Staubli VAL3: RobotMotion3.dtx

bool bSignal
bool bTxt1
bool bTxt2
bool bTxt3
bool btrig
public dio fout = {link=fOut0}
public frame FrmDraw = {x=1000, y=-100, fatherId=world[0]}
mdesc mNomSpeed
num l_nInit = 1500
num nNumTotal = 799
num nNumrecord
num nTxtTotal = 2
num n_sTxt
num ndelay = 258.323
public num nnnn
num ntime = 459.89
pointRx pfrmCad[1500]
  [0] = {x=16.915, y=-25.265, z=273.2, rx=-177, ry=0.5, rz=-161.069, fatherId=FrmDraw[0]}
  [1] = {x=15.593, y=-24.767, z=273.202, rx=-177, ry=0.459, rz=-162.61, fatherId=FrmDraw[0]}
  [2] = {x=14.003, y=-24.227, z=273.204, rx=-177, ry=0.41, rz=-164.442, fatherId=FrmDraw[0]}
  [3] = {x=12.409, y=-23.75, z=273.205, rx=-177, ry=0.362, rz=-166.257, fatherId=FrmDraw[0]}
  [4] = {x=10.813, y=-23.335, z=273.207, rx=-177, ry=0.314, rz=-168.059, fatherId=FrmDraw[0]}
  [5] = {x=9.215, y=-22.978, z=273.208, rx=-177, ry=0.267, rz=-169.848, fatherId=FrmDraw[0]}
  [6] = {x=7.615, y=-22.681, z=273.209, rx=-177, ry=0.22, rz=-171.628, fatherId=FrmDraw[0]}
  [7] = {x=6.014, y=-22.441, z=273.209, rx=-177, ry=0.173, rz=-173.399, fatherId=FrmDraw[0]}
  [8] = {x=4.411, y=-22.259, z=273.21, rx=-177, ry=0.127, rz=-175.164, fatherId=FrmDraw[0]}
  [9] = {x=2.807, y=-22.133, z=273.21, rx=-177, ry=0.081, rz=-176.925, fatherId=FrmDraw[0]}
  [10] = {x=1.203, y=-22.063, z=273.211, rx=-177, ry=0.034, rz=-178.683, fatherId=FrmDraw[0]}
  [11] = {x=0.134, y=-22.047, z=273.211, rx=-177, ry=0.004, rz=-179.854, fatherId=FrmDraw[0]}
  [12] = {x=-1.203, y=-22.063, z=273.211, rx=-177, ry=-0.034, rz=178.683, fatherId=FrmDraw[0]}
  [13] = {x=-2.807, y=-22.133, z=273.21, rx=-177, ry=-0.081, rz=176.925, fatherId=FrmDraw[0]}
  [14] = {x=-4.411, y=-22.259, z=273.21, rx=-177, ry=-0.127, rz=175.164, fatherId=FrmDraw[0]}
  [15] = {x=-6.014, y=-22.441, z=273.209, rx=-177, ry=-0.173, rz=173.399, fatherId=FrmDraw[0]}
  [16] = {x=-7.615, y=-22.681, z=273.209, rx=-177, ry=-0.22, rz=171.628, fatherId=FrmDraw[0]}
  [17] = {x=-9.215, y=-22.978, z=273.208, rx=-177, ry=-0.267, rz=169.848, fatherId=FrmDraw[0]}
  [18] = {x=-10.813, y=-23.335, z=273.207, rx=-177, ry=-0.314, rz=168.059, fatherId=FrmDraw[0]}
  [19] = {x=-12.409, y=-23.75, z=273.205, rx=-177, ry=-0.362, rz=166.257, fatherId=FrmDraw[0]}
  [20] = {x=-14.002, y=-24.227, z=273.204, rx=-177, ry=-0.41, rz=164.442, fatherId=FrmDraw[0]}
  [21] = {x=-15.593, y=-24.767, z=273.202, rx=-177, ry=-0.459, rz=162.61, fatherId=FrmDraw[0]}
  [22] = {x=-16.915, y=-25.265, z=273.2, rx=-177, ry=-0.5, rz=161.069, fatherId=FrmDraw[0]}
  [23] = {x=-16.935, y=-25.265, z=270.798, rx=-177, ry=-0.5, rz=161.071, fatherId=FrmDraw[0]}
  [24] = {x=-16.956, y=-25.264, z=268.2, rx=-177, ry=-0.5, rz=161.073, fatherId=FrmDraw[0]}
  [25] = {x=-15.63, y=-24.766, z=268.202, rx=-177, ry=-0.459, rz=162.614, fatherId=FrmDraw[0]}
  [26] = {x=-14.035, y=-24.226, z=268.204, rx=-177, ry=-0.41, rz=164.445, fatherId=FrmDraw[0]}
  [27] = {x=-12.438, y=-23.75, z=268.205, rx=-177, ry=-0.362, rz=166.26, fatherId=FrmDraw[0]}
  [28] = {x=-10.838, y=-23.334, z=268.207, rx=-177, ry=-0.314, rz=168.061, fatherId=FrmDraw[0]}
  [29] = {x=-9.236, y=-22.978, z=268.208, rx=-177, ry=-0.266, rz=169.85, fatherId=FrmDraw[0]}
  [30] = {x=-7.633, y=-22.681, z=268.209, rx=-177, ry=-0.22, rz=171.63, fatherId=FrmDraw[0]}
  [31] = {x=-6.027, y=-22.441, z=268.209, rx=-177, ry=-0.173, rz=173.401, fatherId=FrmDraw[0]}
  [32] = {x=-4.421, y=-22.259, z=268.21, rx=-177, ry=-0.127, rz=175.165, fatherId=FrmDraw[0]}
  [33] = {x=-2.814, y=-22.133, z=268.21, rx=-177, ry=-0.081, rz=176.926, fatherId=FrmDraw[0]}
  [34] = {x=-1.206, y=-22.063, z=268.211, rx=-177, ry=-0.034, rz=178.683, fatherId=FrmDraw[0]}
  [35] = {x=-0.134, y=-22.047, z=268.211, rx=-177, ry=-0.004, rz=179.854, fatherId=FrmDraw[0]}
  [36] = {x=1.206, y=-22.063, z=268.211, rx=-177, ry=0.034, rz=-178.683, fatherId=FrmDraw[0]}
  [37] = {x=2.814, y=-22.133, z=268.21, rx=-177, ry=0.081, rz=-176.926, fatherId=FrmDraw[0]}
  [38] = {x=4.421, y=-22.259, z=268.21, rx=-177, ry=0.127, rz=-175.165, fatherId=FrmDraw[0]}
  [39] = {x=6.027, y=-22.441, z=268.209, rx=-177, ry=0.173, rz=-173.401, fatherId=FrmDraw[0]}
  [40] = {x=7.633, y=-22.681, z=268.209, rx=-177, ry=0.22, rz=-171.63, fatherId=FrmDraw[0]}
  [41] = {x=9.237, y=-22.978, z=268.208, rx=-177, ry=0.266, rz=-169.85, fatherId=FrmDraw[0]}
  [42] = {x=10.838, y=-23.334, z=268.207, rx=-177, ry=0.314, rz=-168.061, fatherId=FrmDraw[0]}
  [43] = {x=12.438, y=-23.75, z=268.205, rx=-177, ry=0.362, rz=-166.26, fatherId=FrmDraw[0]}
  [44] = {x=14.035, y=-24.226, z=268.204, rx=-177, ry=0.41, rz=-164.445, fatherId=FrmDraw[0]}
  [45] = {x=15.63, y=-24.766, z=268.202, rx=-177, ry=0.459, rz=-162.614, fatherId=FrmDraw[0]}
  [46] = {x=16.956, y=-25.264, z=268.2, rx=-177, ry=0.5, rz=-161.073, fatherId=FrmDraw[0]}
  [47] = {x=16.978, y=-25.265, z=265.798, rx=-177, ry=0.5, rz=-161.071, fatherId=FrmDraw[0]}
  [48] = {x=17.003, y=-25.265, z=263.201, rx=-177, ry=0.5, rz=-161.069, fatherId=FrmDraw[0]}
  [49] = {x=15.673, y=-24.767, z=263.202, rx=-177, ry=0.459, rz=-162.61, fatherId=FrmDraw[0]}
  [50] = {x=14.074, y=-24.227, z=263.204, rx=-177, ry=0.41, rz=-164.442, fatherId=FrmDraw[0]}
  [51] = {x=12.472, y=-23.75, z=263.205, rx=-177, ry=0.362, rz=-166.257, fatherId=FrmDraw[0]}
  [52] = {x=10.868, y=-23.335, z=263.207, rx=-177, ry=0.314, rz=-168.059, fatherId=FrmDraw[0]}
  [53] = {x=9.262, y=-22.978, z=263.208, rx=-177, ry=0.267, rz=-169.848, fatherId=FrmDraw[0]}
  [54] = {x=7.653, y=-22.681, z=263.209, rx=-177, ry=0.22, rz=-171.628, fatherId=FrmDraw[0]}
  [55] = {x=6.044, y=-22.441, z=263.209, rx=-177, ry=0.173, rz=-173.399, fatherId=FrmDraw[0]}
  [56] = {x=4.433, y=-22.259, z=263.21, rx=-177, ry=0.127, rz=-175.164, fatherId=FrmDraw[0]}
  [57] = {x=2.821, y=-22.133, z=263.21, rx=-177, ry=0.081, rz=-176.925, fatherId=FrmDraw[0]}
  [58] = {x=1.209, y=-22.063, z=263.211, rx=-177, ry=0.034, rz=-178.683, fatherId=FrmDraw[0]}
  [59] = {x=0.134, y=-22.047, z=263.211, rx=-177, ry=0.004, rz=-179.854, fatherId=FrmDraw[0]}
  [60] = {x=-1.209, y=-22.063, z=263.211, rx=-177, ry=-0.034, rz=178.683, fatherId=FrmDraw[0]}
  [61] = {x=-2.821, y=-22.133, z=263.21, rx=-177, ry=-0.081, rz=176.925, fatherId=FrmDraw[0]}
  [62] = {x=-4.433, y=-22.259, z=263.21, rx=-177, ry=-0.127, rz=175.165, fatherId=FrmDraw[0]}
  [63] = {x=-6.044, y=-22.441, z=263.209, rx=-177, ry=-0.173, rz=173.399, fatherId=FrmDraw[0]}
  [64] = {x=-7.653, y=-22.681, z=263.209, rx=-177, ry=-0.22, rz=171.628, fatherId=FrmDraw[0]}
  [65] = {x=-9.262, y=-22.978, z=263.208, rx=-177, ry=-0.267, rz=169.848, fatherId=FrmDraw[0]}
  [66] = {x=-10.868, y=-23.335, z=263.207, rx=-177, ry=-0.314, rz=168.059, fatherId=FrmDraw[0]}
  [67] = {x=-12.472, y=-23.75, z=263.205, rx=-177, ry=-0.362, rz=166.257, fatherId=FrmDraw[0]}
  [68] = {x=-14.074, y=-24.227, z=263.204, rx=-177, ry=-0.41, rz=164.442, fatherId=FrmDraw[0]}
  [69] = {x=-15.673, y=-24.767, z=263.202, rx=-177, ry=-0.459, rz=162.61, fatherId=FrmDraw[0]}
  [70] = {x=-17.003, y=-25.265, z=263.201, rx=-177, ry=-0.5, rz=161.069, fatherId=FrmDraw[0]}
  [71] = {x=-17.022, y=-25.265, z=260.799, rx=-177, ry=-0.5, rz=161.071, fatherId=FrmDraw[0]}
  [72] = {x=-17.043, y=-25.264, z=258.201, rx=-177, ry=-0.5, rz=161.074, fatherId=FrmDraw[0]}
  [73] = {x=-15.455, y=-24.676, z=258.203, rx=-177, ry=-0.451, rz=162.906, fatherId=FrmDraw[0]}
  [74] = {x=-13.865, y=-24.15, z=258.204, rx=-177, ry=-0.403, rz=164.72, fatherId=FrmDraw[0]}
  [75] = {x=-12.271, y=-23.686, z=258.206, rx=-177, ry=-0.355, rz=166.519, fatherId=FrmDraw[0]}
  [76] = {x=-10.675, y=-23.282, z=258.207, rx=-177, ry=-0.307, rz=168.304, fatherId=FrmDraw[0]}
  [77] = {x=-9.077, y=-22.937, z=258.208, rx=-177, ry=-0.26, rz=170.078, fatherId=FrmDraw[0]}
  [78] = {x=-7.478, y=-22.649, z=258.209, rx=-177, ry=-0.214, rz=171.842, fatherId=FrmDraw[0]}
  [79] = {x=-5.877, y=-22.418, z=258.209, rx=-177, ry=-0.168, rz=173.599, fatherId=FrmDraw[0]}
  [80] = {x=-4.275, y=-22.243, z=258.21, rx=-177, ry=-0.122, rz=175.349, fatherId=FrmDraw[0]}
  [81] = {x=-2.672, y=-22.123, z=258.21, rx=-177, ry=-0.076, rz=177.095, fatherId=FrmDraw[0]}
  [82] = {x=-1.069, y=-22.059, z=258.211, rx=-177, ry=-0.03, rz=178.838, fatherId=FrmDraw[0]}
  [83] = {y=-22.047, z=258.211, rx=-177, rz=180, fatherId=FrmDraw[0]}
  [84] = {x=1.069, y=-22.059, z=258.211, rx=-177, ry=0.03, rz=-178.838, fatherId=FrmDraw[0]}
  [85] = {x=2.672, y=-22.123, z=258.21, rx=-177, ry=0.076, rz=-177.095, fatherId=FrmDraw[0]}
  [86] = {x=4.275, y=-22.243, z=258.21, rx=-177, ry=0.122, rz=-175.349, fatherId=FrmDraw[0]}
  [87] = {x=5.877, y=-22.418, z=258.209, rx=-177, ry=0.168, rz=-173.599, fatherId=FrmDraw[0]}
  [88] = {x=7.478, y=-22.649, z=258.209, rx=-177, ry=0.214, rz=-171.842, fatherId=FrmDraw[0]}
  [89] = {x=9.077, y=-22.937, z=258.208, rx=-177, ry=0.26, rz=-170.078, fatherId=FrmDraw[0]}
  [90] = {x=10.675, y=-23.282, z=258.207, rx=-177, ry=0.307, rz=-168.304, fatherId=FrmDraw[0]}
  [91] = {x=12.271, y=-23.686, z=258.206, rx=-177, ry=0.355, rz=-166.519, fatherId=FrmDraw[0]}
  [92] = {x=13.865, y=-24.15, z=258.204, rx=-177, ry=0.403, rz=-164.72, fatherId=FrmDraw[0]}
  [93] = {x=15.455, y=-24.676, z=258.203, rx=-177, ry=0.451, rz=-162.906, fatherId=FrmDraw[0]}
  [94] = {x=17.043, y=-25.264, z=258.201, rx=-177, ry=0.5, rz=-161.073, fatherId=FrmDraw[0]}
  [95] = {x=17.066, y=-25.265, z=255.799, rx=-177, ry=0.5, rz=-161.072, fatherId=FrmDraw[0]}
  [96] = {x=17.09, y=-25.265, z=253.201, rx=-177, ry=0.5, rz=-161.07, fatherId=FrmDraw[0]}
  [97] = {x=15.763, y=-24.77, z=253.203, rx=-177, ry=0.459, rz=-162.598, fatherId=FrmDraw[0]}
  [98] = {x=14.169, y=-24.234, z=253.204, rx=-177, ry=0.411, rz=-164.416, fatherId=FrmDraw[0]}
  [99] = {x=12.571, y=-23.76, z=253.206, rx=-177, ry=0.363, rz=-166.217, fatherId=FrmDraw[0]}
  [100] = {x=10.971, y=-23.346, z=253.207, rx=-177, ry=0.315, rz=-168.005, fatherId=FrmDraw[0]}
  [101] = {x=9.369, y=-22.991, z=253.208, rx=-177, ry=0.268, rz=-169.781, fatherId=FrmDraw[0]}
  [102] = {x=7.765, y=-22.693, z=253.209, rx=-177, ry=0.222, rz=-171.547, fatherId=FrmDraw[0]}
  [103] = {x=6.16, y=-22.453, z=253.209, rx=-177, ry=0.176, rz=-173.305, fatherId=FrmDraw[0]}
  [104] = {x=4.554, y=-22.268, z=253.21, rx=-177, ry=0.13, rz=-175.057, fatherId=FrmDraw[0]}
  [105] = {x=2.947, y=-22.139, z=253.21, rx=-177, ry=0.084, rz=-176.804, fatherId=FrmDraw[0]}
  [106] = {x=1.34, y=-22.066, z=253.211, rx=-177, ry=0.038, rz=-178.548, fatherId=FrmDraw[0]}
  [107] = {x=0.268, y=-22.048, z=253.211, rx=-177, ry=0.008, rz=-179.71, fatherId=FrmDraw[0]}
  [108] = {x=-1.34, y=-22.066, z=253.211, rx=-177, ry=-0.038, rz=178.548, fatherId=FrmDraw[0]}
  [109] = {x=-2.947, y=-22.139, z=253.21, rx=-177, ry=-0.084, rz=176.804, fatherId=FrmDraw[0]}
  [110] = {x=-4.554, y=-22.268, z=253.21, rx=-177, ry=-0.13, rz=175.057, fatherId=FrmDraw[0]}
  [111] = {x=-6.16, y=-22.453, z=253.209, rx=-177, ry=-0.176, rz=173.305, fatherId=FrmDraw[0]}
  [112] = {x=-7.765, y=-22.693, z=253.209, rx=-177, ry=-0.222, rz=171.547, fatherId=FrmDraw[0]}
  [113] = {x=-9.369, y=-22.991, z=253.208, rx=-177, ry=-0.268, rz=169.781, fatherId=FrmDraw[0]}
  [114] = {x=-10.971, y=-23.346, z=253.207, rx=-177, ry=-0.315, rz=168.005, fatherId=FrmDraw[0]}
  [115] = {x=-12.571, y=-23.76, z=253.206, rx=-177, ry=-0.363, rz=166.217, fatherId=FrmDraw[0]}
  [116] = {x=-14.169, y=-24.234, z=253.204, rx=-177, ry=-0.411, rz=164.416, fatherId=FrmDraw[0]}
  [117] = {x=-15.763, y=-24.77, z=253.203, rx=-177, ry=-0.459, rz=162.598, fatherId=FrmDraw[0]}
  [118] = {x=-17.09, y=-25.265, z=253.201, rx=-177, ry=-0.5, rz=161.07, fatherId=FrmDraw[0]}
  [119] = {x=-17.109, y=-25.265, z=250.799, rx=-177, ry=-0.5, rz=161.071, fatherId=FrmDraw[0]}
  [120] = {x=-17.13, y=-25.264, z=248.201, rx=-177, ry=-0.5, rz=161.074, fatherId=FrmDraw[0]}
  [121] = {x=-15.8, y=-24.769, z=248.203, rx=-177, ry=-0.459, rz=162.602, fatherId=FrmDraw[0]}
  [122] = {x=-14.202, y=-24.234, z=248.204, rx=-177, ry=-0.411, rz=164.419, fatherId=FrmDraw[0]}
  [123] = {x=-12.6, y=-23.76, z=248.206, rx=-177, ry=-0.363, rz=166.22, fatherId=FrmDraw[0]}
  [124] = {x=-10.996, y=-23.346, z=248.207, rx=-177, ry=-0.315, rz=168.007, fatherId=FrmDraw[0]}
  [125] = {x=-9.391, y=-22.99, z=248.208, rx=-177, ry=-0.268, rz=169.783, fatherId=FrmDraw[0]}
  [126] = {x=-7.783, y=-22.693, z=248.209, rx=-177, ry=-0.222, rz=171.549, fatherId=FrmDraw[0]}
  [127] = {x=-6.174, y=-22.453, z=248.209, rx=-177, ry=-0.175, rz=173.306, fatherId=FrmDraw[0]}
  [128] = {x=-4.565, y=-22.268, z=248.21, rx=-177, ry=-0.13, rz=175.058, fatherId=FrmDraw[0]}
  [129] = {x=-2.954, y=-22.139, z=248.21, rx=-177, ry=-0.084, rz=176.804, fatherId=FrmDraw[0]}
  [130] = {x=-1.343, y=-22.066, z=248.211, rx=-177, ry=-0.038, rz=178.548, fatherId=FrmDraw[0]}
  [131] = {y=-22.047, z=248.211, rx=-177, rz=180, fatherId=FrmDraw[0]}
  [132] = {x=1.343, y=-22.066, z=248.211, rx=-177, ry=0.038, rz=-178.548, fatherId=FrmDraw[0]}
  [133] = {x=2.954, y=-22.139, z=248.21, rx=-177, ry=0.084, rz=-176.804, fatherId=FrmDraw[0]}
  [134] = {x=4.565, y=-22.268, z=248.21, rx=-177, ry=0.13, rz=-175.058, fatherId=FrmDraw[0]}
  [135] = {x=6.174, y=-22.453, z=248.209, rx=-177, ry=0.175, rz=-173.306, fatherId=FrmDraw[0]}
  [136] = {x=7.783, y=-22.693, z=248.209, rx=-177, ry=0.222, rz=-171.549, fatherId=FrmDraw[0]}
  [137] = {x=9.391, y=-22.99, z=248.208, rx=-177, ry=0.268, rz=-169.783, fatherId=FrmDraw[0]}
  [138] = {x=10.997, y=-23.346, z=248.207, rx=-177, ry=0.315, rz=-168.007, fatherId=FrmDraw[0]}
  [139] = {x=12.6, y=-23.76, z=248.206, rx=-177, ry=0.363, rz=-166.22, fatherId=FrmDraw[0]}
  [140] = {x=14.202, y=-24.234, z=248.204, rx=-177, ry=0.411, rz=-164.419, fatherId=FrmDraw[0]}
  [141] = {x=15.8, y=-24.769, z=248.203, rx=-177, ry=0.459, rz=-162.602, fatherId=FrmDraw[0]}
  [142] = {x=17.13, y=-25.264, z=248.201, rx=-177, ry=0.5, rz=-161.074, fatherId=FrmDraw[0]}
  [143] = {x=17.153, y=-25.265, z=245.799, rx=-177, ry=0.5, rz=-161.072, fatherId=FrmDraw[0]}
  [144] = {x=17.177, y=-25.265, z=243.201, rx=-177, ry=0.5, rz=-161.07, fatherId=FrmDraw[0]}
  [145] = {x=15.589, y=-24.681, z=243.203, rx=-177, ry=0.451, rz=-162.888, fatherId=FrmDraw[0]}
  [146] = {x=13.998, y=-24.159, z=243.205, rx=-177, ry=0.403, rz=-164.689, fatherId=FrmDraw[0]}
  [147] = {x=12.404, y=-23.697, z=243.206, rx=-177, ry=0.356, rz=-166.474, fatherId=FrmDraw[0]}
  [148] = {x=10.808, y=-23.294, z=243.207, rx=-177, ry=0.309, rz=-168.247, fatherId=FrmDraw[0]}
  [149] = {x=9.21, y=-22.95, z=243.208, rx=-177, ry=0.262, rz=-170.007, fatherId=FrmDraw[0]}
  [150] = {x=7.61, y=-22.661, z=243.209, rx=-177, ry=0.216, rz=-171.759, fatherId=FrmDraw[0]}
  [151] = {x=6.01, y=-22.429, z=243.21, rx=-177, ry=0.17, rz=-173.502, fatherId=FrmDraw[0]}
  [152] = {x=4.408, y=-22.252, z=243.21, rx=-177, ry=0.125, rz=-175.24, fatherId=FrmDraw[0]}
  [153] = {x=2.805, y=-22.13, z=243.21, rx=-177, ry=0.079, rz=-176.973, fatherId=FrmDraw[0]}
  [154] = {x=1.202, y=-22.062, z=243.211, rx=-177, ry=0.034, rz=-178.703, fatherId=FrmDraw[0]}
  [155] = {x=0.134, y=-22.047, z=243.211, rx=-177, ry=0.004, rz=-179.856, fatherId=FrmDraw[0]}
  [156] = {x=-1.202, y=-22.062, z=243.211, rx=-177, ry=-0.034, rz=178.703, fatherId=FrmDraw[0]}
  [157] = {x=-2.805, y=-22.13, z=243.21, rx=-177, ry=-0.079, rz=176.973, fatherId=FrmDraw[0]}
  [158] = {x=-4.408, y=-22.252, z=243.21, rx=-177, ry=-0.125, rz=175.24, fatherId=FrmDraw[0]}
  [159] = {x=-6.01, y=-22.429, z=243.21, rx=-177, ry=-0.17, rz=173.502, fatherId=FrmDraw[0]}
  [160] = {x=-7.61, y=-22.661, z=243.209, rx=-177, ry=-0.216, rz=171.759, fatherId=FrmDraw[0]}
  [161] = {x=-9.21, y=-22.95, z=243.208, rx=-177, ry=-0.262, rz=170.007, fatherId=FrmDraw[0]}
  [162] = {x=-10.808, y=-23.294, z=243.207, rx=-177, ry=-0.309, rz=168.247, fatherId=FrmDraw[0]}
  [163] = {x=-12.404, y=-23.697, z=243.206, rx=-177, ry=-0.356, rz=166.474, fatherId=FrmDraw[0]}
  [164] = {x=-13.998, y=-24.159, z=243.205, rx=-177, ry=-0.403, rz=164.689, fatherId=FrmDraw[0]}
  [165] = {x=-15.589, y=-24.681, z=243.203, rx=-177, ry=-0.451, rz=162.888, fatherId=FrmDraw[0]}
  [166] = {x=-17.177, y=-25.265, z=243.201, rx=-177, ry=-0.5, rz=161.07, fatherId=FrmDraw[0]}
  [167] = {x=-17.197, y=-25.265, z=240.799, rx=-177, ry=-0.5, rz=161.072, fatherId=FrmDraw[0]}
  [168] = {x=-17.218, y=-25.264, z=238.202, rx=-177, ry=-0.5, rz=161.074, fatherId=FrmDraw[0]}
  [169] = {x=-15.625, y=-24.68, z=238.203, rx=-177, ry=-0.451, rz=162.892, fatherId=FrmDraw[0]}
  [170] = {x=-14.03, y=-24.158, z=238.205, rx=-177, ry=-0.403, rz=164.692, fatherId=FrmDraw[0]}
  [171] = {x=-12.433, y=-23.696, z=238.206, rx=-177, ry=-0.356, rz=166.477, fatherId=FrmDraw[0]}
  [172] = {x=-10.833, y=-23.294, z=238.207, rx=-177, ry=-0.309, rz=168.249, fatherId=FrmDraw[0]}
  [173] = {x=-9.231, y=-22.949, z=238.208, rx=-177, ry=-0.262, rz=170.009, fatherId=FrmDraw[0]}
  [174] = {x=-7.628, y=-22.661, z=238.209, rx=-177, ry=-0.216, rz=171.76, fatherId=FrmDraw[0]}
  [175] = {x=-6.023, y=-22.429, z=238.21, rx=-177, ry=-0.17, rz=173.503, fatherId=FrmDraw[0]}
  [176] = {x=-4.418, y=-22.252, z=238.21, rx=-177, ry=-0.125, rz=175.241, fatherId=FrmDraw[0]}
  [177] = {x=-2.812, y=-22.13, z=238.21, rx=-177, ry=-0.079, rz=176.973, fatherId=FrmDraw[0]}
  [178] = {x=-1.205, y=-22.062, z=238.211, rx=-177, ry=-0.034, rz=178.703, fatherId=FrmDraw[0]}
  [179] = {x=-0.134, y=-22.047, z=238.211, rx=-177, ry=-0.004, rz=179.856, fatherId=FrmDraw[0]}
  [180] = {x=1.205, y=-22.062, z=238.211, rx=-177, ry=0.034, rz=-178.703, fatherId=FrmDraw[0]}
  [181] = {x=2.812, y=-22.13, z=238.21, rx=-177, ry=0.079, rz=-176.973, fatherId=FrmDraw[0]}
  [182] = {x=4.418, y=-22.252, z=238.21, rx=-177, ry=0.125, rz=-175.241, fatherId=FrmDraw[0]}
  [183] = {x=6.023, y=-22.429, z=238.21, rx=-177, ry=0.17, rz=-173.503, fatherId=FrmDraw[0]}
  [184] = {x=7.628, y=-22.661, z=238.209, rx=-177, ry=0.216, rz=-171.76, fatherId=FrmDraw[0]}
  [185] = {x=9.231, y=-22.949, z=238.208, rx=-177, ry=0.262, rz=-170.009, fatherId=FrmDraw[0]}
  [186] = {x=10.833, y=-23.294, z=238.207, rx=-177, ry=0.309, rz=-168.249, fatherId=FrmDraw[0]}
  [187] = {x=12.433, y=-23.697, z=238.206, rx=-177, ry=0.356, rz=-166.477, fatherId=FrmDraw[0]}
  [188] = {x=14.03, y=-24.158, z=238.205, rx=-177, ry=0.403, rz=-164.692, fatherId=FrmDraw[0]}
  [189] = {x=15.625, y=-24.68, z=238.203, rx=-177, ry=0.451, rz=-162.892, fatherId=FrmDraw[0]}
  [190] = {x=17.218, y=-25.264, z=238.202, rx=-177, ry=0.5, rz=-161.074, fatherId=FrmDraw[0]}
  [191] = {x=17.24, y=-25.265, z=235.8, rx=-177, ry=0.5, rz=-161.072, fatherId=FrmDraw[0]}
  [192] = {x=17.265, y=-25.265, z=233.202, rx=-177, ry=0.5, rz=-161.07, fatherId=FrmDraw[0]}
  [193] = {x=15.934, y=-24.774, z=233.203, rx=-177, ry=0.46, rz=-162.586, fatherId=FrmDraw[0]}
  [194] = {x=14.335, y=-24.242, z=233.205, rx=-177, ry=0.411, rz=-164.39, fatherId=FrmDraw[0]}
  [195] = {x=12.733, y=-23.77, z=233.206, rx=-177, ry=0.364, rz=-166.178, fatherId=FrmDraw[0]}
  [196] = {x=11.129, y=-23.358, z=233.207, rx=-177, ry=0.317, rz=-167.952, fatherId=FrmDraw[0]}
  [197] = {x=9.524, y=-23.003, z=233.208, rx=-177, ry=0.27, rz=-169.715, fatherId=FrmDraw[0]}
  [198] = {x=7.916, y=-22.706, z=233.209, rx=-177, ry=0.224, rz=-171.467, fatherId=FrmDraw[0]}
  [199] = {x=6.308, y=-22.464, z=233.209, rx=-177, ry=0.178, rz=-173.212, fatherId=FrmDraw[0]}
  [200] = {x=4.698, y=-22.278, z=233.21, rx=-177, ry=0.132, rz=-174.95, fatherId=FrmDraw[0]}
  [201] = {x=3.088, y=-22.147, z=233.21, rx=-177, ry=0.087, rz=-176.684, fatherId=FrmDraw[0]}
  [202] = {x=1.477, y=-22.07, z=233.211, rx=-177, ry=0.042, rz=-178.415, fatherId=FrmDraw[0]}
  [203] = {x=0.134, y=-22.047, z=233.211, rx=-177, ry=0.004, rz=-179.856, fatherId=FrmDraw[0]}
  [204] = {x=-1.477, y=-22.07, z=233.211, rx=-177, ry=-0.042, rz=178.415, fatherId=FrmDraw[0]}
  [205] = {x=-3.088, y=-22.147, z=233.21, rx=-177, ry=-0.087, rz=176.684, fatherId=FrmDraw[0]}
  [206] = {x=-4.698, y=-22.278, z=233.21, rx=-177, ry=-0.132, rz=174.95, fatherId=FrmDraw[0]}
  [207] = {x=-6.308, y=-22.464, z=233.209, rx=-177, ry=-0.178, rz=173.212, fatherId=FrmDraw[0]}
  [208] = {x=-7.916, y=-22.706, z=233.209, rx=-177, ry=-0.224, rz=171.467, fatherId=FrmDraw[0]}
  [209] = {x=-9.524, y=-23.003, z=233.208, rx=-177, ry=-0.27, rz=169.715, fatherId=FrmDraw[0]}
  [210] = {x=-11.129, y=-23.358, z=233.207, rx=-177, ry=-0.317, rz=167.952, fatherId=FrmDraw[0]}
  [211] = {x=-12.733, y=-23.77, z=233.206, rx=-177, ry=-0.364, rz=166.178, fatherId=FrmDraw[0]}
  [212] = {x=-14.335, y=-24.242, z=233.205, rx=-177, ry=-0.411, rz=164.39, fatherId=FrmDraw[0]}
  [213] = {x=-15.934, y=-24.774, z=233.203, rx=-177, ry=-0.46, rz=162.586, fatherId=FrmDraw[0]}
  [214] = {x=-17.265, y=-25.265, z=233.202, rx=-177, ry=-0.5, rz=161.07, fatherId=FrmDraw[0]}
  [215] = {x=-17.284, y=-25.265, z=230.8, rx=-177, ry=-0.5, rz=161.072, fatherId=FrmDraw[0]}
  [216] = {x=-17.305, y=-25.264, z=228.202, rx=-177, ry=-0.5, rz=161.074, fatherId=FrmDraw[0]}
  [217] = {x=-15.971, y=-24.773, z=228.203, rx=-177, ry=-0.459, rz=162.59, fatherId=FrmDraw[0]}
  [218] = {x=-14.368, y=-24.241, z=228.205, rx=-177, ry=-0.411, rz=164.393, fatherId=FrmDraw[0]}
  [219] = {x=-12.762, y=-23.769, z=228.206, rx=-177, ry=-0.364, rz=166.181, fatherId=FrmDraw[0]}
  [220] = {x=-11.155, y=-23.357, z=228.207, rx=-177, ry=-0.317, rz=167.955, fatherId=FrmDraw[0]}
  [221] = {x=-9.545, y=-23.003, z=228.208, rx=-177, ry=-0.27, rz=169.717, fatherId=FrmDraw[0]}
  [222] = {x=-7.934, y=-22.705, z=228.209, rx=-177, ry=-0.224, rz=171.469, fatherId=FrmDraw[0]}
  [223] = {x=-6.322, y=-22.464, z=228.209, rx=-177, ry=-0.178, rz=173.213, fatherId=FrmDraw[0]}
  [224] = {x=-4.709, y=-22.278, z=228.21, rx=-177, ry=-0.132, rz=174.951, fatherId=FrmDraw[0]}
  [225] = {x=-3.095, y=-22.146, z=228.21, rx=-177, ry=-0.087, rz=176.685, fatherId=FrmDraw[0]}
  [226] = {x=-1.48, y=-22.07, z=228.211, rx=-177, ry=-0.042, rz=178.415, fatherId=FrmDraw[0]}
  [227] = {x=-0.135, y=-22.047, z=228.211, rx=-177, ry=-0.004, rz=179.856, fatherId=FrmDraw[0]}
  [228] = {x=1.48, y=-22.07, z=228.211, rx=-177, ry=0.042, rz=-178.415, fatherId=FrmDraw[0]}
  [229] = {x=3.095, y=-22.146, z=228.21, rx=-177, ry=0.087, rz=-176.685, fatherId=FrmDraw[0]}
  [230] = {x=4.709, y=-22.278, z=228.21, rx=-177, ry=0.132, rz=-174.951, fatherId=FrmDraw[0]}
  [231] = {x=6.322, y=-22.464, z=228.209, rx=-177, ry=0.178, rz=-173.213, fatherId=FrmDraw[0]}
  [232] = {x=7.934, y=-22.705, z=228.209, rx=-177, ry=0.224, rz=-171.469, fatherId=FrmDraw[0]}
  [233] = {x=9.545, y=-23.003, z=228.208, rx=-177, ry=0.27, rz=-169.717, fatherId=FrmDraw[0]}
  [234] = {x=11.155, y=-23.357, z=228.207, rx=-177, ry=0.317, rz=-167.955, fatherId=FrmDraw[0]}
  [235] = {x=12.763, y=-23.769, z=228.206, rx=-177, ry=0.364, rz=-166.181, fatherId=FrmDraw[0]}
  [236] = {x=14.368, y=-24.241, z=228.205, rx=-177, ry=0.411, rz=-164.393, fatherId=FrmDraw[0]}
  [237] = {x=15.971, y=-24.773, z=228.203, rx=-177, ry=0.459, rz=-162.59, fatherId=FrmDraw[0]}
  [238] = {x=17.305, y=-25.264, z=228.202, rx=-177, ry=0.5, rz=-161.074, fatherId=FrmDraw[0]}
  [239] = {x=17.328, y=-25.264, z=225.8, rx=-177, ry=0.5, rz=-161.072, fatherId=FrmDraw[0]}
  [240] = {x=17.352, y=-25.265, z=223.202, rx=-177, ry=0.5, rz=-161.07, fatherId=FrmDraw[0]}
  [241] = {x=15.759, y=-24.685, z=223.204, rx=-177, ry=0.452, rz=-162.874, fatherId=FrmDraw[0]}
  [242] = {x=14.163, y=-24.166, z=223.205, rx=-177, ry=0.404, rz=-164.662, fatherId=FrmDraw[0]}
  [243] = {x=12.565, y=-23.707, z=223.206, rx=-177, ry=0.357, rz=-166.434, fatherId=FrmDraw[0]}
  [244] = {x=10.965, y=-23.306, z=223.207, rx=-177, ry=0.31, rz=-168.192, fatherId=FrmDraw[0]}
  [245] = {x=9.364, y=-22.962, z=223.208, rx=-177, ry=0.264, rz=-169.94, fatherId=FrmDraw[0]}
  [246] = {x=7.761, y=-22.673, z=223.209, rx=-177, ry=0.218, rz=-171.678, fatherId=FrmDraw[0]}
  [247] = {x=6.156, y=-22.44, z=223.21, rx=-177, ry=0.173, rz=-173.409, fatherId=FrmDraw[0]}
  [248] = {x=4.551, y=-22.261, z=223.21, rx=-177, ry=0.128, rz=-175.133, fatherId=FrmDraw[0]}
  [249] = {x=2.945, y=-22.137, z=223.21, rx=-177, ry=0.082, rz=-176.853, fatherId=FrmDraw[0]}
  [250] = {x=1.339, y=-22.065, z=223.211, rx=-177, ry=0.037, rz=-178.57, fatherId=FrmDraw[0]}
  [251] = {x=0.268, y=-22.048, z=223.211, rx=-177, ry=0.007, rz=-179.714, fatherId=FrmDraw[0]}
  [252] = {x=-1.339, y=-22.065, z=223.211, rx=-177, ry=-0.037, rz=178.57, fatherId=FrmDraw[0]}
  [253] = {x=-2.945, y=-22.137, z=223.21, rx=-177, ry=-0.082, rz=176.853, fatherId=FrmDraw[0]}
  [254] = {x=-4.551, y=-22.261, z=223.21, rx=-177, ry=-0.128, rz=175.133, fatherId=FrmDraw[0]}
  [255] = {x=-6.156, y=-22.44, z=223.21, rx=-177, ry=-0.173, rz=173.409, fatherId=FrmDraw[0]}
  [256] = {x=-7.761, y=-22.673, z=223.209, rx=-177, ry=-0.218, rz=171.678, fatherId=FrmDraw[0]}
  [257] = {x=-9.364, y=-22.962, z=223.208, rx=-177, ry=-0.264, rz=169.94, fatherId=FrmDraw[0]}
  [258] = {x=-10.965, y=-23.306, z=223.207, rx=-177, ry=-0.31, rz=168.192, fatherId=FrmDraw[0]}
  [259] = {x=-12.565, y=-23.707, z=223.206, rx=-177, ry=-0.357, rz=166.434, fatherId=FrmDraw[0]}
  [260] = {x=-14.163, y=-24.166, z=223.205, rx=-177, ry=-0.404, rz=164.662, fatherId=FrmDraw[0]}
  [261] = {x=-15.759, y=-24.685, z=223.204, rx=-177, ry=-0.452, rz=162.874, fatherId=FrmDraw[0]}
  [262] = {x=-17.352, y=-25.265, z=223.202, rx=-177, ry=-0.5, rz=161.07, fatherId=FrmDraw[0]}
  [263] = {x=-17.371, y=-25.265, z=220.8, rx=-177, ry=-0.5, rz=161.072, fatherId=FrmDraw[0]}
  [264] = {x=-17.392, y=-25.264, z=218.202, rx=-177, ry=-0.5, rz=161.074, fatherId=FrmDraw[0]}
  [265] = {x=-15.795, y=-24.684, z=218.204, rx=-177, ry=-0.452, rz=162.878, fatherId=FrmDraw[0]}
  [266] = {x=-14.196, y=-24.166, z=218.205, rx=-177, ry=-0.404, rz=164.665, fatherId=FrmDraw[0]}
  [267] = {x=-12.594, y=-23.706, z=218.206, rx=-177, ry=-0.357, rz=166.436, fatherId=FrmDraw[0]}
  [268] = {x=-10.99, y=-23.305, z=218.207, rx=-177, ry=-0.31, rz=168.195, fatherId=FrmDraw[0]}
  [269] = {x=-9.385, y=-22.961, z=218.208, rx=-177, ry=-0.264, rz=169.942, fatherId=FrmDraw[0]}
  [270] = {x=-7.778, y=-22.673, z=218.209, rx=-177, ry=-0.218, rz=171.68, fatherId=FrmDraw[0]}
  [271] = {x=-6.17, y=-22.44, z=218.21, rx=-177, ry=-0.173, rz=173.41, fatherId=FrmDraw[0]}
  [272] = {x=-4.561, y=-22.261, z=218.21, rx=-177, ry=-0.128, rz=175.134, fatherId=FrmDraw[0]}
  [273] = {x=-2.952, y=-22.137, z=218.21, rx=-177, ry=-0.082, rz=176.854, fatherId=FrmDraw[0]}
  [274] = {x=-1.342, y=-22.065, z=218.211, rx=-177, ry=-0.037, rz=178.57, fatherId=FrmDraw[0]}
  [275] = {y=-22.047, z=218.211, rx=-177, rz=180, fatherId=FrmDraw[0]}
  [276] = {x=1.342, y=-22.065, z=218.211, rx=-177, ry=0.037, rz=-178.57, fatherId=FrmDraw[0]}
  [277] = {x=2.952, y=-22.137, z=218.21, rx=-177, ry=0.082, rz=-176.854, fatherId=FrmDraw[0]}
  [278] = {x=4.561, y=-22.261, z=218.21, rx=-177, ry=0.128, rz=-175.134, fatherId=FrmDraw[0]}
  [279] = {x=6.17, y=-22.44, z=218.21, rx=-177, ry=0.173, rz=-173.41, fatherId=FrmDraw[0]}
  [280] = {x=7.778, y=-22.673, z=218.209, rx=-177, ry=0.218, rz=-171.68, fatherId=FrmDraw[0]}
  [281] = {x=9.385, y=-22.961, z=218.208, rx=-177, ry=0.264, rz=-169.942, fatherId=FrmDraw[0]}
  [282] = {x=10.99, y=-23.305, z=218.207, rx=-177, ry=0.31, rz=-168.195, fatherId=FrmDraw[0]}
  [283] = {x=12.594, y=-23.706, z=218.206, rx=-177, ry=0.357, rz=-166.436, fatherId=FrmDraw[0]}
  [284] = {x=14.196, y=-24.166, z=218.205, rx=-177, ry=0.404, rz=-164.665, fatherId=FrmDraw[0]}
  [285] = {x=15.795, y=-24.684, z=218.204, rx=-177, ry=0.452, rz=-162.878, fatherId=FrmDraw[0]}
  [286] = {x=17.392, y=-25.264, z=218.202, rx=-177, ry=0.5, rz=-161.074, fatherId=FrmDraw[0]}
  [287] = {x=17.415, y=-25.264, z=215.8, rx=-177, ry=0.5, rz=-161.072, fatherId=FrmDraw[0]}
  [288] = {x=17.439, y=-25.265, z=213.203, rx=-177, ry=0.5, rz=-161.07, fatherId=FrmDraw[0]}
  [289] = {x=15.838, y=-24.685, z=213.204, rx=-177, ry=0.452, rz=-162.874, fatherId=FrmDraw[0]}
  [290] = {x=14.234, y=-24.166, z=213.205, rx=-177, ry=0.404, rz=-164.662, fatherId=FrmDraw[0]}
  [291] = {x=12.628, y=-23.707, z=213.206, rx=-177, ry=0.357, rz=-166.434, fatherId=FrmDraw[0]}
  [292] = {x=11.02, y=-23.306, z=213.207, rx=-177, ry=0.31, rz=-168.192, fatherId=FrmDraw[0]}
  [293] = {x=9.41, y=-22.962, z=213.208, rx=-177, ry=0.264, rz=-169.94, fatherId=FrmDraw[0]}
  [294] = {x=7.799, y=-22.673, z=213.209, rx=-177, ry=0.218, rz=-171.678, fatherId=FrmDraw[0]}
  [295] = {x=6.186, y=-22.44, z=213.21, rx=-177, ry=0.173, rz=-173.409, fatherId=FrmDraw[0]}
  [296] = {x=4.573, y=-22.261, z=213.21, rx=-177, ry=0.128, rz=-175.133, fatherId=FrmDraw[0]}
  [297] = {x=2.959, y=-22.137, z=213.21, rx=-177, ry=0.082, rz=-176.853, fatherId=FrmDraw[0]}
  [298] = {x=1.345, y=-22.065, z=213.211, rx=-177, ry=0.037, rz=-178.57, fatherId=FrmDraw[0]}
  [299] = {x=0.269, y=-22.048, z=213.211, rx=-177, ry=0.007, rz=-179.714, fatherId=FrmDraw[0]}
  [300] = {x=-1.345, y=-22.065, z=213.211, rx=-177, ry=-0.037, rz=178.57, fatherId=FrmDraw[0]}
  [301] = {x=-2.959, y=-22.137, z=213.21, rx=-177, ry=-0.082, rz=176.853, fatherId=FrmDraw[0]}
  [302] = {x=-4.573, y=-22.261, z=213.21, rx=-177, ry=-0.128, rz=175.133, fatherId=FrmDraw[0]}
  [303] = {x=-6.186, y=-22.44, z=213.21, rx=-177, ry=-0.173, rz=173.409, fatherId=FrmDraw[0]}
  [304] = {x=-7.799, y=-22.673, z=213.209, rx=-177, ry=-0.218, rz=171.678, fatherId=FrmDraw[0]}
  [305] = {x=-9.41, y=-22.962, z=213.208, rx=-177, ry=-0.264, rz=169.94, fatherId=FrmDraw[0]}
  [306] = {x=-11.02, y=-23.306, z=213.207, rx=-177, ry=-0.31, rz=168.192, fatherId=FrmDraw[0]}
  [307] = {x=-12.628, y=-23.707, z=213.206, rx=-177, ry=-0.357, rz=166.434, fatherId=FrmDraw[0]}
  [308] = {x=-14.234, y=-24.166, z=213.205, rx=-177, ry=-0.404, rz=164.662, fatherId=FrmDraw[0]}
  [309] = {x=-15.838, y=-24.685, z=213.204, rx=-177, ry=-0.452, rz=162.874, fatherId=FrmDraw[0]}
  [310] = {x=-17.439, y=-25.265, z=213.203, rx=-177, ry=-0.5, rz=161.07, fatherId=FrmDraw[0]}
  [311] = {x=-17.459, y=-25.264, z=210.801, rx=-177, ry=-0.5, rz=161.072, fatherId=FrmDraw[0]}
  [312] = {x=-17.48, y=-25.264, z=208.203, rx=-177, ry=-0.5, rz=161.074, fatherId=FrmDraw[0]}
  [313] = {x=-16.142, y=-24.776, z=208.204, rx=-177, ry=-0.46, rz=162.579, fatherId=FrmDraw[0]}
  [314] = {x=-14.535, y=-24.248, z=208.205, rx=-177, ry=-0.412, rz=164.368, fatherId=FrmDraw[0]}
  [315] = {x=-12.925, y=-23.779, z=208.206, rx=-177, ry=-0.365, rz=166.142, fatherId=FrmDraw[0]}
  [316] = {x=-11.313, y=-23.368, z=208.207, rx=-177, ry=-0.318, rz=167.903, fatherId=FrmDraw[0]}
  [317] = {x=-9.7, y=-23.015, z=208.208, rx=-177, ry=-0.272, rz=169.652, fatherId=FrmDraw[0]}
  [318] = {x=-8.085, y=-22.717, z=208.209, rx=-177, ry=-0.226, rz=171.391, fatherId=FrmDraw[0]}
  [319] = {x=-6.47, y=-22.475, z=208.21, rx=-177, ry=-0.18, rz=173.122, fatherId=FrmDraw[0]}
  [320] = {x=-4.853, y=-22.287, z=208.21, rx=-177, ry=-0.135, rz=174.847, fatherId=FrmDraw[0]}
  [321] = {x=-3.236, y=-22.154, z=208.21, rx=-177, ry=-0.09, rz=176.567, fatherId=FrmDraw[0]}
  [322] = {x=-1.618, y=-22.074, z=208.211, rx=-177, ry=-0.045, rz=178.284, fatherId=FrmDraw[0]}
  [323] = {y=-22.047, z=208.211, rx=-177, rz=180, fatherId=FrmDraw[0]}
  [324] = {x=1.618, y=-22.074, z=208.211, rx=-177, ry=0.045, rz=-178.284, fatherId=FrmDraw[0]}
  [325] = {x=3.236, y=-22.154, z=208.21, rx=-177, ry=0.09, rz=-176.567, fatherId=FrmDraw[0]}
  [326] = {x=4.853, y=-22.287, z=208.21, rx=-177, ry=0.135, rz=-174.847, fatherId=FrmDraw[0]}
  [327] = {x=6.47, y=-22.475, z=208.21, rx=-177, ry=0.18, rz=-173.122, fatherId=FrmDraw[0]}
  [328] = {x=8.085, y=-22.717, z=208.209, rx=-177, ry=0.226, rz=-171.391, fatherId=FrmDraw[0]}
  [329] = {x=9.7, y=-23.015, z=208.208, rx=-177, ry=0.272, rz=-169.651, fatherId=FrmDraw[0]}
  [330] = {x=11.313, y=-23.368, z=208.207, rx=-177, ry=0.318, rz=-167.902, fatherId=FrmDraw[0]}
  [331] = {x=12.925, y=-23.779, z=208.206, rx=-177, ry=0.365, rz=-166.142, fatherId=FrmDraw[0]}
  [332] = {x=14.535, y=-24.248, z=208.205, rx=-177, ry=0.412, rz=-164.368, fatherId=FrmDraw[0]}
  [333] = {x=16.142, y=-24.776, z=208.204, rx=-177, ry=0.46, rz=-162.579, fatherId=FrmDraw[0]}
  [334] = {x=17.48, y=-25.264, z=208.203, rx=-177, ry=0.5, rz=-161.074, fatherId=FrmDraw[0]}
  [335] = {x=17.502, y=-25.264, z=205.801, rx=-177, ry=0.5, rz=-161.072, fatherId=FrmDraw[0]}
  [336] = {x=17.527, y=-25.265, z=203.203, rx=-177, ry=0.5, rz=-161.07, fatherId=FrmDraw[0]}
  [337] = {x=15.929, y=-24.689, z=203.204, rx=-177, ry=0.452, rz=-162.861, fatherId=FrmDraw[0]}
  [338] = {x=14.329, y=-24.174, z=203.206, rx=-177, ry=0.405, rz=-164.635, fatherId=FrmDraw[0]}
  [339] = {x=12.727, y=-23.717, z=203.207, rx=-177, ry=0.358, rz=-166.393, fatherId=FrmDraw[0]}
  [340] = {x=11.123, y=-23.317, z=203.208, rx=-177, ry=0.312, rz=-168.139, fatherId=FrmDraw[0]}
  [341] = {x=9.518, y=-22.974, z=203.208, rx=-177, ry=0.266, rz=-169.874, fatherId=FrmDraw[0]}
  [342] = {x=7.911, y=-22.685, z=203.209, rx=-177, ry=0.22, rz=-171.599, fatherId=FrmDraw[0]}
  [343] = {x=6.303, y=-22.451, z=203.21, rx=-177, ry=0.175, rz=-173.316, fatherId=FrmDraw[0]}
  [344] = {x=4.695, y=-22.271, z=203.21, rx=-177, ry=0.13, rz=-175.028, fatherId=FrmDraw[0]}
  [345] = {x=3.085, y=-22.144, z=203.21, rx=-177, ry=0.086, rz=-176.735, fatherId=FrmDraw[0]}
  [346] = {x=1.476, y=-22.069, z=203.211, rx=-177, ry=0.041, rz=-178.439, fatherId=FrmDraw[0]}
  [347] = {x=0.134, y=-22.047, z=203.211, rx=-177, ry=0.004, rz=-179.858, fatherId=FrmDraw[0]}
  [348] = {x=-1.476, y=-22.069, z=203.211, rx=-177, ry=-0.041, rz=178.439, fatherId=FrmDraw[0]}
  [349] = {x=-3.085, y=-22.144, z=203.21, rx=-177, ry=-0.086, rz=176.735, fatherId=FrmDraw[0]}
  [350] = {x=-4.695, y=-22.271, z=203.21, rx=-177, ry=-0.13, rz=175.028, fatherId=FrmDraw[0]}
  [351] = {x=-6.303, y=-22.451, z=203.21, rx=-177, ry=-0.175, rz=173.316, fatherId=FrmDraw[0]}
  [352] = {x=-7.911, y=-22.685, z=203.209, rx=-177, ry=-0.22, rz=171.599, fatherId=FrmDraw[0]}
  [353] = {x=-9.518, y=-22.974, z=203.208, rx=-177, ry=-0.266, rz=169.874, fatherId=FrmDraw[0]}
  [354] = {x=-11.123, y=-23.317, z=203.208, rx=-177, ry=-0.312, rz=168.139, fatherId=FrmDraw[0]}
  [355] = {x=-12.727, y=-23.717, z=203.207, rx=-177, ry=-0.358, rz=166.393, fatherId=FrmDraw[0]}
  [356] = {x=-14.329, y=-24.174, z=203.206, rx=-177, ry=-0.405, rz=164.635, fatherId=FrmDraw[0]}
  [357] = {x=-15.929, y=-24.689, z=203.204, rx=-177, ry=-0.452, rz=162.861, fatherId=FrmDraw[0]}
  [358] = {x=-17.527, y=-25.265, z=203.203, rx=-177, ry=-0.5, rz=161.07, fatherId=FrmDraw[0]}
  [359] = {x=-17.546, y=-25.264, z=200.801, rx=-177, ry=-0.5, rz=161.072, fatherId=FrmDraw[0]}
  [360] = {x=-17.567, y=-25.264, z=198.203, rx=-177, ry=-0.5, rz=161.074, fatherId=FrmDraw[0]}
  [361] = {x=-15.966, y=-24.688, z=198.204, rx=-177, ry=-0.452, rz=162.864, fatherId=FrmDraw[0]}
  [362] = {x=-14.362, y=-24.173, z=198.206, rx=-177, ry=-0.405, rz=164.638, fatherId=FrmDraw[0]}
  [363] = {x=-12.756, y=-23.716, z=198.207, rx=-177, ry=-0.358, rz=166.396, fatherId=FrmDraw[0]}
  [364] = {x=-11.148, y=-23.317, z=198.208, rx=-177, ry=-0.312, rz=168.141, fatherId=FrmDraw[0]}
  [365] = {x=-9.539, y=-22.973, z=198.208, rx=-177, ry=-0.266, rz=169.876, fatherId=FrmDraw[0]}
  [366] = {x=-7.929, y=-22.685, z=198.209, rx=-177, ry=-0.22, rz=171.6, fatherId=FrmDraw[0]}
  [367] = {x=-6.317, y=-22.451, z=198.21, rx=-177, ry=-0.175, rz=173.318, fatherId=FrmDraw[0]}
  [368] = {x=-4.705, y=-22.271, z=198.21, rx=-177, ry=-0.13, rz=175.029, fatherId=FrmDraw[0]}
  [369] = {x=-3.092, y=-22.143, z=198.21, rx=-177, ry=-0.086, rz=176.736, fatherId=FrmDraw[0]}
  [370] = {x=-1.479, y=-22.069, z=198.211, rx=-177, ry=-0.041, rz=178.439, fatherId=FrmDraw[0]}
  [371] = {x=-0.134, y=-22.047, z=198.211, rx=-177, ry=-0.004, rz=179.858, fatherId=FrmDraw[0]}
  [372] = {x=1.479, y=-22.069, z=198.211, rx=-177, ry=0.041, rz=-178.439, fatherId=FrmDraw[0]}
  [373] = {x=3.092, y=-22.143, z=198.21, rx=-177, ry=0.086, rz=-176.736, fatherId=FrmDraw[0]}
  [374] = {x=4.705, y=-22.271, z=198.21, rx=-177, ry=0.13, rz=-175.029, fatherId=FrmDraw[0]}
  [375] = {x=6.317, y=-22.451, z=198.21, rx=-177, ry=0.175, rz=-173.318, fatherId=FrmDraw[0]}
  [376] = {x=7.929, y=-22.685, z=198.209, rx=-177, ry=0.22, rz=-171.6, fatherId=FrmDraw[0]}
  [377] = {x=9.539, y=-22.973, z=198.208, rx=-177, ry=0.266, rz=-169.875, fatherId=FrmDraw[0]}
  [378] = {x=11.148, y=-23.317, z=198.208, rx=-177, ry=0.312, rz=-168.141, fatherId=FrmDraw[0]}
  [379] = {x=12.756, y=-23.716, z=198.207, rx=-177, ry=0.358, rz=-166.396, fatherId=FrmDraw[0]}
  [380] = {x=14.362, y=-24.173, z=198.206, rx=-177, ry=0.405, rz=-164.638, fatherId=FrmDraw[0]}
  [381] = {x=15.966, y=-24.688, z=198.204, rx=-177, ry=0.452, rz=-162.864, fatherId=FrmDraw[0]}
  [382] = {x=17.567, y=-25.264, z=198.203, rx=-177, ry=0.5, rz=-161.074, fatherId=FrmDraw[0]}
  [383] = {x=17.59, y=-25.264, z=195.801, rx=-177, ry=0.5, rz=-161.072, fatherId=FrmDraw[0]}
  [384] = {x=17.614, y=-25.265, z=193.203, rx=-177, ry=0.5, rz=-161.07, fatherId=FrmDraw[0]}
  [385] = {x=16.008, y=-24.689, z=193.205, rx=-177, ry=0.452, rz=-162.861, fatherId=FrmDraw[0]}
  [386] = {x=14.4, y=-24.174, z=193.206, rx=-177, ry=0.405, rz=-164.635, fatherId=FrmDraw[0]}
  [387] = {x=12.79, y=-23.717, z=193.207, rx=-177, ry=0.358, rz=-166.393, fatherId=FrmDraw[0]}
  [388] = {x=11.178, y=-23.317, z=193.208, rx=-177, ry=0.312, rz=-168.139, fatherId=FrmDraw[0]}
  [389] = {x=9.564, y=-22.974, z=193.209, rx=-177, ry=0.266, rz=-169.874, fatherId=FrmDraw[0]}
  [390] = {x=7.949, y=-22.685, z=193.209, rx=-177, ry=0.22, rz=-171.599, fatherId=FrmDraw[0]}
  [391] = {x=6.334, y=-22.451, z=193.21, rx=-177, ry=0.175, rz=-173.316, fatherId=FrmDraw[0]}
  [392] = {x=4.717, y=-22.271, z=193.21, rx=-177, ry=0.13, rz=-175.028, fatherId=FrmDraw[0]}
  [393] = {x=3.1, y=-22.143, z=193.21, rx=-177, ry=0.086, rz=-176.735, fatherId=FrmDraw[0]}
  [394] = {x=1.483, y=-22.069, z=193.211, rx=-177, ry=0.041, rz=-178.439, fatherId=FrmDraw[0]}
  [395] = {x=0.135, y=-22.047, z=193.211, rx=-177, ry=0.004, rz=-179.858, fatherId=FrmDraw[0]}
  [396] = {x=-1.483, y=-22.069, z=193.211, rx=-177, ry=-0.041, rz=178.439, fatherId=FrmDraw[0]}
  [397] = {x=-3.1, y=-22.144, z=193.21, rx=-177, ry=-0.086, rz=176.735, fatherId=FrmDraw[0]}
  [398] = {x=-4.717, y=-22.271, z=193.21, rx=-177, ry=-0.13, rz=175.028, fatherId=FrmDraw[0]}
  [399] = {x=-6.334, y=-22.451, z=193.21, rx=-177, ry=-0.175, rz=173.316, fatherId=FrmDraw[0]}
  [400] = {x=-7.949, y=-22.685, z=193.209, rx=-177, ry=-0.22, rz=171.599, fatherId=FrmDraw[0]}
  [401] = {x=-9.564, y=-22.974, z=193.209, rx=-177, ry=-0.266, rz=169.874, fatherId=FrmDraw[0]}
  [402] = {x=-11.178, y=-23.317, z=193.208, rx=-177, ry=-0.312, rz=168.139, fatherId=FrmDraw[0]}
  [403] = {x=-12.79, y=-23.717, z=193.207, rx=-177, ry=-0.358, rz=166.393, fatherId=FrmDraw[0]}
  [404] = {x=-14.4, y=-24.174, z=193.206, rx=-177, ry=-0.405, rz=164.635, fatherId=FrmDraw[0]}
  [405] = {x=-16.008, y=-24.689, z=193.205, rx=-177, ry=-0.452, rz=162.861, fatherId=FrmDraw[0]}
  [406] = {x=-17.614, y=-25.265, z=193.203, rx=-177, ry=-0.5, rz=161.07, fatherId=FrmDraw[0]}
  [407] = {x=-17.633, y=-25.264, z=190.801, rx=-177, ry=-0.5, rz=161.072, fatherId=FrmDraw[0]}
  [408] = {x=-17.654, y=-25.264, z=188.204, rx=-177, ry=-0.5, rz=161.074, fatherId=FrmDraw[0]}
  [409] = {x=-16.057, y=-24.692, z=188.205, rx=-177, ry=-0.452, rz=162.851, fatherId=FrmDraw[0]}
  [410] = {x=-14.457, y=-24.18, z=188.206, rx=-177, ry=-0.405, rz=164.611, fatherId=FrmDraw[0]}
  [411] = {x=-12.855, y=-23.726, z=188.207, rx=-177, ry=-0.359, rz=166.356, fatherId=FrmDraw[0]}
  [412] = {x=-11.252, y=-23.328, z=188.208, rx=-177, ry=-0.313, rz=168.089, fatherId=FrmDraw[0]}
  [413] = {x=-9.647, y=-22.985, z=188.209, rx=-177, ry=-0.268, rz=169.81, fatherId=FrmDraw[0]}
  [414] = {x=-8.041, y=-22.697, z=188.209, rx=-177, ry=-0.222, rz=171.522, fatherId=FrmDraw[0]}
  [415] = {x=-6.434, y=-22.462, z=188.21, rx=-177, ry=-0.178, rz=173.227, fatherId=FrmDraw[0]}
  [416] = {x=-4.826, y=-22.28, z=188.21, rx=-177, ry=-0.133, rz=174.925, fatherId=FrmDraw[0]}
  [417] = {x=-3.218, y=-22.15, z=188.21, rx=-177, ry=-0.089, rz=176.619, fatherId=FrmDraw[0]}
  [418] = {x=-1.609, y=-22.073, z=188.211, rx=-177, ry=-0.044, rz=178.31, fatherId=FrmDraw[0]}
  [419] = {y=-22.047, z=188.211, rx=-177, rz=180, fatherId=FrmDraw[0]}
  [420] = {x=1.609, y=-22.073, z=188.211, rx=-177, ry=0.044, rz=-178.31, fatherId=FrmDraw[0]}
  [421] = {x=3.218, y=-22.15, z=188.21, rx=-177, ry=0.089, rz=-176.619, fatherId=FrmDraw[0]}
  [422] = {x=4.826, y=-22.28, z=188.21, rx=-177, ry=0.133, rz=-174.925, fatherId=FrmDraw[0]}
  [423] = {x=6.434, y=-22.462, z=188.21, rx=-177, ry=0.178, rz=-173.227, fatherId=FrmDraw[0]}
  [424] = {x=8.041, y=-22.697, z=188.209, rx=-177, ry=0.222, rz=-171.522, fatherId=FrmDraw[0]}
  [425] = {x=9.647, y=-22.985, z=188.209, rx=-177, ry=0.268, rz=-169.81, fatherId=FrmDraw[0]}
  [426] = {x=11.252, y=-23.328, z=188.208, rx=-177, ry=0.313, rz=-168.089, fatherId=FrmDraw[0]}
  [427] = {x=12.855, y=-23.726, z=188.207, rx=-177, ry=0.359, rz=-166.356, fatherId=FrmDraw[0]}
  [428] = {x=14.457, y=-24.18, z=188.206, rx=-177, ry=0.405, rz=-164.611, fatherId=FrmDraw[0]}
  [429] = {x=16.057, y=-24.692, z=188.205, rx=-177, ry=0.452, rz=-162.851, fatherId=FrmDraw[0]}
  [430] = {x=17.654, y=-25.264, z=188.204, rx=-177, ry=0.5, rz=-161.074, fatherId=FrmDraw[0]}
  [431] = {x=17.677, y=-25.264, z=185.801, rx=-177, ry=0.5, rz=-161.072, fatherId=FrmDraw[0]}
  [432] = {x=17.702, y=-25.265, z=183.204, rx=-177, ry=0.5, rz=-161.07, fatherId=FrmDraw[0]}
  [433] = {x=16.099, y=-24.693, z=183.205, rx=-177, ry=0.453, rz=-162.847, fatherId=FrmDraw[0]}
  [434] = {x=14.495, y=-24.181, z=183.206, rx=-177, ry=0.406, rz=-164.608, fatherId=FrmDraw[0]}
  [435] = {x=12.889, y=-23.727, z=183.207, rx=-177, ry=0.359, rz=-166.354, fatherId=FrmDraw[0]}
  [436] = {x=11.281, y=-23.329, z=183.208, rx=-177, ry=0.313, rz=-168.086, fatherId=FrmDraw[0]}
  [437] = {x=9.672, y=-22.986, z=183.209, rx=-177, ry=0.268, rz=-169.808, fatherId=FrmDraw[0]}
  [438] = {x=8.062, y=-22.697, z=183.209, rx=-177, ry=0.222, rz=-171.521, fatherId=FrmDraw[0]}
  [439] = {x=6.45, y=-22.462, z=183.21, rx=-177, ry=0.178, rz=-173.225, fatherId=FrmDraw[0]}
  [440] = {x=4.839, y=-22.28, z=183.21, rx=-177, ry=0.133, rz=-174.924, fatherId=FrmDraw[0]}
  [441] = {x=3.226, y=-22.151, z=183.21, rx=-177, ry=0.089, rz=-176.619, fatherId=FrmDraw[0]}
  [442] = {x=1.613, y=-22.073, z=183.211, rx=-177, ry=0.044, rz=-178.31, fatherId=FrmDraw[0]}
  [443] = {y=-22.047, z=183.211, rx=-177, rz=180, fatherId=FrmDraw[0]}
  [444] = {x=-1.613, y=-22.073, z=183.211, rx=-177, ry=-0.044, rz=178.31, fatherId=FrmDraw[0]}
  [445] = {x=-3.226, y=-22.151, z=183.21, rx=-177, ry=-0.089, rz=176.619, fatherId=FrmDraw[0]}
  [446] = {x=-4.838, y=-22.28, z=183.21, rx=-177, ry=-0.133, rz=174.924, fatherId=FrmDraw[0]}
  [447] = {x=-6.45, y=-22.462, z=183.21, rx=-177, ry=-0.178, rz=173.225, fatherId=FrmDraw[0]}
  [448] = {x=-8.062, y=-22.697, z=183.209, rx=-177, ry=-0.222, rz=171.521, fatherId=FrmDraw[0]}
  [449] = {x=-9.672, y=-22.986, z=183.209, rx=-177, ry=-0.268, rz=169.808, fatherId=FrmDraw[0]}
  [450] = {x=-11.281, y=-23.329, z=183.208, rx=-177, ry=-0.313, rz=168.086, fatherId=FrmDraw[0]}
  [451] = {x=-12.889, y=-23.727, z=183.207, rx=-177, ry=-0.359, rz=166.354, fatherId=FrmDraw[0]}
  [452] = {x=-14.495, y=-24.181, z=183.206, rx=-177, ry=-0.406, rz=164.608, fatherId=FrmDraw[0]}
  [453] = {x=-16.099, y=-24.693, z=183.205, rx=-177, ry=-0.453, rz=162.847, fatherId=FrmDraw[0]}
  [454] = {x=-17.701, y=-25.265, z=183.204, rx=-177, ry=-0.5, rz=161.07, fatherId=FrmDraw[0]}
  [455] = {x=-17.721, y=-25.264, z=180.802, rx=-177, ry=-0.5, rz=161.072, fatherId=FrmDraw[0]}
  [456] = {x=-17.742, y=-25.264, z=178.204, rx=-177, ry=-0.5, rz=161.074, fatherId=FrmDraw[0]}
  [457] = {x=-16.136, y=-24.692, z=178.205, rx=-177, ry=-0.452, rz=162.851, fatherId=FrmDraw[0]}
  [458] = {x=-14.528, y=-24.18, z=178.206, rx=-177, ry=-0.405, rz=164.611, fatherId=FrmDraw[0]}
  [459] = {x=-12.918, y=-23.726, z=178.207, rx=-177, ry=-0.359, rz=166.356, fatherId=FrmDraw[0]}
  [460] = {x=-11.306, y=-23.328, z=178.208, rx=-177, ry=-0.313, rz=168.089, fatherId=FrmDraw[0]}
  [461] = {x=-9.693, y=-22.985, z=178.209, rx=-177, ry=-0.268, rz=169.81, fatherId=FrmDraw[0]}
  [462] = {x=-8.08, y=-22.697, z=178.209, rx=-177, ry=-0.222, rz=171.522, fatherId=FrmDraw[0]}
  [463] = {x=-6.465, y=-22.462, z=178.21, rx=-177, ry=-0.178, rz=173.227, fatherId=FrmDraw[0]}
  [464] = {x=-4.849, y=-22.28, z=178.21, rx=-177, ry=-0.133, rz=174.925, fatherId=FrmDraw[0]}
  [465] = {x=-3.233, y=-22.15, z=178.21, rx=-177, ry=-0.089, rz=176.619, fatherId=FrmDraw[0]}
  [466] = {x=-1.617, y=-22.073, z=178.211, rx=-177, ry=-0.044, rz=178.31, fatherId=FrmDraw[0]}
  [467] = {y=-22.047, z=178.211, rx=-177, rz=180, fatherId=FrmDraw[0]}
  [468] = {x=1.617, y=-22.073, z=178.211, rx=-177, ry=0.044, rz=-178.31, fatherId=FrmDraw[0]}
  [469] = {x=3.233, y=-22.15, z=178.21, rx=-177, ry=0.089, rz=-176.619, fatherId=FrmDraw[0]}
  [470] = {x=4.849, y=-22.28, z=178.21, rx=-177, ry=0.133, rz=-174.925, fatherId=FrmDraw[0]}
  [471] = {x=6.465, y=-22.462, z=178.21, rx=-177, ry=0.178, rz=-173.227, fatherId=FrmDraw[0]}
  [472] = {x=8.08, y=-22.697, z=178.209, rx=-177, ry=0.222, rz=-171.522, fatherId=FrmDraw[0]}
  [473] = {x=9.694, y=-22.985, z=178.209, rx=-177, ry=0.268, rz=-169.81, fatherId=FrmDraw[0]}
  [474] = {x=11.306, y=-23.328, z=178.208, rx=-177, ry=0.313, rz=-168.089, fatherId=FrmDraw[0]}
  [475] = {x=12.918, y=-23.726, z=178.207, rx=-177, ry=0.359, rz=-166.356, fatherId=FrmDraw[0]}
  [476] = {x=14.528, y=-24.18, z=178.206, rx=-177, ry=0.405, rz=-164.611, fatherId=FrmDraw[0]}
  [477] = {x=16.136, y=-24.692, z=178.205, rx=-177, ry=0.452, rz=-162.851, fatherId=FrmDraw[0]}
  [478] = {x=17.742, y=-25.264, z=178.204, rx=-177, ry=0.5, rz=-161.074, fatherId=FrmDraw[0]}
  [479] = {x=17.764, y=-25.264, z=175.802, rx=-177, ry=0.5, rz=-161.072, fatherId=FrmDraw[0]}
  [480] = {x=17.789, y=-25.265, z=173.204, rx=-177, ry=0.5, rz=-161.07, fatherId=FrmDraw[0]}
  [481] = {x=16.178, y=-24.693, z=173.205, rx=-177, ry=0.453, rz=-162.848, fatherId=FrmDraw[0]}
  [482] = {x=14.566, y=-24.181, z=173.206, rx=-177, ry=0.406, rz=-164.608, fatherId=FrmDraw[0]}
  [483] = {x=12.952, y=-23.727, z=173.207, rx=-177, ry=0.359, rz=-166.354, fatherId=FrmDraw[0]}
  [484] = {x=11.336, y=-23.329, z=173.208, rx=-177, ry=0.313, rz=-168.086, fatherId=FrmDraw[0]}
  [485] = {x=9.719, y=-22.986, z=173.209, rx=-177, ry=0.268, rz=-169.808, fatherId=FrmDraw[0]}
  [486] = {x=8.101, y=-22.697, z=173.209, rx=-177, ry=0.222, rz=-171.521, fatherId=FrmDraw[0]}
  [487] = {x=6.481, y=-22.462, z=173.21, rx=-177, ry=0.178, rz=-173.225, fatherId=FrmDraw[0]}
  [488] = {x=4.862, y=-22.28, z=173.21, rx=-177, ry=0.133, rz=-174.924, fatherId=FrmDraw[0]}
  [489] = {x=3.241, y=-22.15, z=173.21, rx=-177, ry=0.089, rz=-176.619, fatherId=FrmDraw[0]}
  [490] = {x=1.621, y=-22.073, z=173.211, rx=-177, ry=0.044, rz=-178.31, fatherId=FrmDraw[0]}
  [491] = {y=-22.047, z=173.211, rx=-177, rz=180, fatherId=FrmDraw[0]}
  [492] = {x=-1.621, y=-22.073, z=173.211, rx=-177, ry=-0.044, rz=178.31, fatherId=FrmDraw[0]}
  [493] = {x=-3.241, y=-22.151, z=173.21, rx=-177, ry=-0.089, rz=176.619, fatherId=FrmDraw[0]}
  [494] = {x=-4.862, y=-22.28, z=173.21, rx=-177, ry=-0.133, rz=174.924, fatherId=FrmDraw[0]}
  [495] = {x=-6.481, y=-22.462, z=173.21, rx=-177, ry=-0.178, rz=173.225, fatherId=FrmDraw[0]}
  [496] = {x=-8.101, y=-22.697, z=173.209, rx=-177, ry=-0.222, rz=171.521, fatherId=FrmDraw[0]}
  [497] = {x=-9.719, y=-22.986, z=173.209, rx=-177, ry=-0.268, rz=169.808, fatherId=FrmDraw[0]}
  [498] = {x=-11.336, y=-23.329, z=173.208, rx=-177, ry=-0.313, rz=168.086, fatherId=FrmDraw[0]}
  [499] = {x=-12.952, y=-23.727, z=173.207, rx=-177, ry=-0.359, rz=166.354, fatherId=FrmDraw[0]}
  [500] = {x=-14.566, y=-24.181, z=173.206, rx=-177, ry=-0.406, rz=164.608, fatherId=FrmDraw[0]}
  [501] = {x=-16.178, y=-24.693, z=173.205, rx=-177, ry=-0.453, rz=162.848, fatherId=FrmDraw[0]}
  [502] = {x=-17.789, y=-25.265, z=173.204, rx=-177, ry=-0.5, rz=161.07, fatherId=FrmDraw[0]}
  [503] = {x=-17.808, y=-25.264, z=170.802, rx=-177, ry=-0.5, rz=161.072, fatherId=FrmDraw[0]}
  [504] = {x=-17.829, y=-25.264, z=168.204, rx=-177, ry=-0.5, rz=161.074, fatherId=FrmDraw[0]}
  [505] = {x=-16.227, y=-24.696, z=168.205, rx=-177, ry=-0.453, rz=162.838, fatherId=FrmDraw[0]}
  [506] = {x=-14.623, y=-24.188, z=168.206, rx=-177, ry=-0.406, rz=164.585, fatherId=FrmDraw[0]}
  [507] = {x=-13.017, y=-23.736, z=168.207, rx=-177, ry=-0.36, rz=166.317, fatherId=FrmDraw[0]}
  [508] = {x=-11.41, y=-23.339, z=168.208, rx=-177, ry=-0.314, rz=168.037, fatherId=FrmDraw[0]}
  [509] = {x=-9.801, y=-22.997, z=168.209, rx=-177, ry=-0.269, rz=169.746, fatherId=FrmDraw[0]}
  [510] = {x=-8.192, y=-22.709, z=168.209, rx=-177, ry=-0.224, rz=171.445, fatherId=FrmDraw[0]}
  [511] = {x=-6.581, y=-22.473, z=168.21, rx=-177, ry=-0.18, rz=173.137, fatherId=FrmDraw[0]}
  [512] = {x=-4.97, y=-22.29, z=168.21, rx=-177, ry=-0.136, rz=174.823, fatherId=FrmDraw[0]}
  [513] = {x=-3.358, y=-22.158, z=168.21, rx=-177, ry=-0.092, rz=176.505, fatherId=FrmDraw[0]}
  [514] = {x=-1.746, y=-22.077, z=168.211, rx=-177, ry=-0.048, rz=178.183, fatherId=FrmDraw[0]}
  [515] = {x=-0.672, y=-22.051, z=168.211, rx=-177, ry=-0.018, rz=179.301, fatherId=FrmDraw[0]}
  [516] = {x=0.134, y=-22.047, z=168.211, rx=-177, ry=0.004, rz=-179.86, fatherId=FrmDraw[0]}
  [517] = {x=1.747, y=-22.077, z=168.211, rx=-177, ry=0.048, rz=-178.183, fatherId=FrmDraw[0]}
  [518] = {x=3.358, y=-22.158, z=168.21, rx=-177, ry=0.092, rz=-176.505, fatherId=FrmDraw[0]}
  [519] = {x=4.97, y=-22.29, z=168.21, rx=-177, ry=0.136, rz=-174.823, fatherId=FrmDraw[0]}
  [520] = {x=6.581, y=-22.473, z=168.21, rx=-177, ry=0.18, rz=-173.137, fatherId=FrmDraw[0]}
  [521] = {x=8.192, y=-22.709, z=168.209, rx=-177, ry=0.224, rz=-171.445, fatherId=FrmDraw[0]}
  [522] = {x=9.801, y=-22.997, z=168.209, rx=-177, ry=0.269, rz=-169.746, fatherId=FrmDraw[0]}
  [523] = {x=11.41, y=-23.339, z=168.208, rx=-177, ry=0.314, rz=-168.037, fatherId=FrmDraw[0]}
  [524] = {x=13.017, y=-23.736, z=168.207, rx=-177, ry=0.36, rz=-166.317, fatherId=FrmDraw[0]}
  [525] = {x=14.623, y=-24.188, z=168.206, rx=-177, ry=0.406, rz=-164.585, fatherId=FrmDraw[0]}
  [526] = {x=16.227, y=-24.696, z=168.205, rx=-177, ry=0.453, rz=-162.838, fatherId=FrmDraw[0]}
  [527] = {x=17.829, y=-25.264, z=168.204, rx=-177, ry=0.5, rz=-161.074, fatherId=FrmDraw[0]}
  [528] = {x=17.852, y=-25.264, z=165.802, rx=-177, ry=0.5, rz=-161.072, fatherId=FrmDraw[0]}
  [529] = {x=17.876, y=-25.265, z=163.204, rx=-177, ry=0.5, rz=-161.07, fatherId=FrmDraw[0]}
  [530] = {x=16.27, y=-24.697, z=163.206, rx=-177, ry=0.453, rz=-162.834, fatherId=FrmDraw[0]}
  [531] = {x=14.661, y=-24.188, z=163.207, rx=-177, ry=0.406, rz=-164.582, fatherId=FrmDraw[0]}
  [532] = {x=13.051, y=-23.736, z=163.207, rx=-177, ry=0.36, rz=-166.314, fatherId=FrmDraw[0]}
  [533] = {x=11.439, y=-23.34, z=163.208, rx=-177, ry=0.314, rz=-168.034, fatherId=FrmDraw[0]}
  [534] = {x=9.827, y=-22.998, z=163.209, rx=-177, ry=0.269, rz=-169.744, fatherId=FrmDraw[0]}
  [535] = {x=8.213, y=-22.709, z=163.209, rx=-177, ry=0.224, rz=-171.444, fatherId=FrmDraw[0]}
  [536] = {x=6.598, y=-22.473, z=163.21, rx=-177, ry=0.18, rz=-173.136, fatherId=FrmDraw[0]}
  [537] = {x=4.983, y=-22.29, z=163.21, rx=-177, ry=0.136, rz=-174.822, fatherId=FrmDraw[0]}
  [538] = {x=3.367, y=-22.158, z=163.21, rx=-177, ry=0.092, rz=-176.504, fatherId=FrmDraw[0]}
  [539] = {x=1.751, y=-22.077, z=163.211, rx=-177, ry=0.048, rz=-178.183, fatherId=FrmDraw[0]}
  [540] = {x=0.673, y=-22.051, z=163.211, rx=-177, ry=0.018, rz=-179.301, fatherId=FrmDraw[0]}
  [541] = {x=-0.135, y=-22.047, z=163.211, rx=-177, ry=-0.004, rz=179.86, fatherId=FrmDraw[0]}
  [542] = {x=-1.751, y=-22.077, z=163.211, rx=-177, ry=-0.048, rz=178.183, fatherId=FrmDraw[0]}
  [543] = {x=-3.367, y=-22.158, z=163.21, rx=-177, ry=-0.092, rz=176.504, fatherId=FrmDraw[0]}
  [544] = {x=-4.983, y=-22.29, z=163.21, rx=-177, ry=-0.136, rz=174.822, fatherId=FrmDraw[0]}
  [545] = {x=-6.598, y=-22.473, z=163.21, rx=-177, ry=-0.18, rz=173.136, fatherId=FrmDraw[0]}
  [546] = {x=-8.213, y=-22.709, z=163.209, rx=-177, ry=-0.224, rz=171.444, fatherId=FrmDraw[0]}
  [547] = {x=-9.827, y=-22.998, z=163.209, rx=-177, ry=-0.269, rz=169.744, fatherId=FrmDraw[0]}
  [548] = {x=-11.439, y=-23.34, z=163.208, rx=-177, ry=-0.314, rz=168.034, fatherId=FrmDraw[0]}
  [549] = {x=-13.051, y=-23.736, z=163.207, rx=-177, ry=-0.36, rz=166.314, fatherId=FrmDraw[0]}
  [550] = {x=-14.661, y=-24.188, z=163.207, rx=-177, ry=-0.406, rz=164.582, fatherId=FrmDraw[0]}
  [551] = {x=-16.27, y=-24.697, z=163.206, rx=-177, ry=-0.453, rz=162.834, fatherId=FrmDraw[0]}
  [552] = {x=-17.876, y=-25.265, z=163.204, rx=-177, ry=-0.5, rz=161.07, fatherId=FrmDraw[0]}
  [553] = {x=-17.896, y=-25.264, z=160.802, rx=-177, ry=-0.5, rz=161.072, fatherId=FrmDraw[0]}
  [554] = {x=-17.917, y=-25.264, z=158.205, rx=-177, ry=-0.5, rz=161.074, fatherId=FrmDraw[0]}
  [555] = {x=-16.306, y=-24.696, z=158.206, rx=-177, ry=-0.453, rz=162.838, fatherId=FrmDraw[0]}
  [556] = {x=-14.694, y=-24.188, z=158.207, rx=-177, ry=-0.406, rz=164.585, fatherId=FrmDraw[0]}
  [557] = {x=-13.08, y=-23.736, z=158.208, rx=-177, ry=-0.36, rz=166.317, fatherId=FrmDraw[0]}
  [558] = {x=-11.465, y=-23.339, z=158.208, rx=-177, ry=-0.314, rz=168.037, fatherId=FrmDraw[0]}
  [559] = {x=-9.848, y=-22.997, z=158.209, rx=-177, ry=-0.269, rz=169.746, fatherId=FrmDraw[0]}
  [560] = {x=-8.231, y=-22.709, z=158.209, rx=-177, ry=-0.224, rz=171.445, fatherId=FrmDraw[0]}
  [561] = {x=-6.613, y=-22.473, z=158.21, rx=-177, ry=-0.18, rz=173.137, fatherId=FrmDraw[0]}
  [562] = {x=-4.994, y=-22.29, z=158.21, rx=-177, ry=-0.136, rz=174.823, fatherId=FrmDraw[0]}
  [563] = {x=-3.374, y=-22.158, z=158.21, rx=-177, ry=-0.092, rz=176.505, fatherId=FrmDraw[0]}
  [564] = {x=-1.755, y=-22.077, z=158.211, rx=-177, ry=-0.048, rz=178.183, fatherId=FrmDraw[0]}
  [565] = {x=-0.675, y=-22.051, z=158.211, rx=-177, ry=-0.018, rz=179.301, fatherId=FrmDraw[0]}
  [566] = {x=0.135, y=-22.047, z=158.211, rx=-177, ry=0.004, rz=-179.86, fatherId=FrmDraw[0]}
  [567] = {x=1.755, y=-22.077, z=158.211, rx=-177, ry=0.048, rz=-178.183, fatherId=FrmDraw[0]}
  [568] = {x=3.374, y=-22.158, z=158.21, rx=-177, ry=0.092, rz=-176.505, fatherId=FrmDraw[0]}
  [569] = {x=4.994, y=-22.29, z=158.21, rx=-177, ry=0.136, rz=-174.823, fatherId=FrmDraw[0]}
  [570] = {x=6.613, y=-22.473, z=158.21, rx=-177, ry=0.18, rz=-173.137, fatherId=FrmDraw[0]}
  [571] = {x=8.231, y=-22.709, z=158.209, rx=-177, ry=0.224, rz=-171.445, fatherId=FrmDraw[0]}
  [572] = {x=9.848, y=-22.997, z=158.209, rx=-177, ry=0.269, rz=-169.746, fatherId=FrmDraw[0]}
  [573] = {x=11.465, y=-23.339, z=158.208, rx=-177, ry=0.314, rz=-168.037, fatherId=FrmDraw[0]}
  [574] = {x=13.08, y=-23.736, z=158.208, rx=-177, ry=0.36, rz=-166.317, fatherId=FrmDraw[0]}
  [575] = {x=14.694, y=-24.188, z=158.207, rx=-177, ry=0.406, rz=-164.585, fatherId=FrmDraw[0]}
  [576] = {x=16.306, y=-24.696, z=158.206, rx=-177, ry=0.453, rz=-162.838, fatherId=FrmDraw[0]}
  [577] = {x=17.917, y=-25.264, z=158.205, rx=-177, ry=0.5, rz=-161.074, fatherId=FrmDraw[0]}
  [578] = {x=17.939, y=-25.264, z=155.803, rx=-177, ry=0.5, rz=-161.072, fatherId=FrmDraw[0]}
  [579] = {x=17.964, y=-25.265, z=153.205, rx=-177, ry=0.5, rz=-161.07, fatherId=FrmDraw[0]}
  [580] = {x=16.361, y=-24.701, z=153.206, rx=-177, ry=0.453, rz=-162.821, fatherId=FrmDraw[0]}
  [581] = {x=14.756, y=-24.196, z=153.207, rx=-177, ry=0.407, rz=-164.556, fatherId=FrmDraw[0]}
  [582] = {x=13.15, y=-23.746, z=153.208, rx=-177, ry=0.361, rz=-166.276, fatherId=FrmDraw[0]}
  [583] = {x=11.543, y=-23.351, z=153.208, rx=-177, ry=0.316, rz=-167.983, fatherId=FrmDraw[0]}
  [584] = {x=9.934, y=-23.01, z=153.209, rx=-177, ry=0.271, rz=-169.68, fatherId=FrmDraw[0]}
  [585] = {x=8.325, y=-22.721, z=153.209, rx=-177, ry=0.226, rz=-171.368, fatherId=FrmDraw[0]}
  [586] = {x=6.714, y=-22.484, z=153.21, rx=-177, ry=0.182, rz=-173.048, fatherId=FrmDraw[0]}
  [587] = {x=5.103, y=-22.299, z=153.21, rx=-177, ry=0.138, rz=-174.722, fatherId=FrmDraw[0]}
  [588] = {x=3.492, y=-22.165, z=153.21, rx=-177, ry=0.095, rz=-176.391, fatherId=FrmDraw[0]}
  [589] = {x=1.88, y=-22.081, z=153.211, rx=-177, ry=0.051, rz=-178.058, fatherId=FrmDraw[0]}
  [590] = {x=0.806, y=-22.053, z=153.211, rx=-177, ry=0.022, rz=-179.168, fatherId=FrmDraw[0]}
  [591] = {x=-0.269, y=-22.048, z=153.211, rx=-177, ry=-0.007, rz=179.723, fatherId=FrmDraw[0]}
  [592] = {x=-1.88, y=-22.081, z=153.211, rx=-177, ry=-0.051, rz=178.058, fatherId=FrmDraw[0]}
  [593] = {x=-3.492, y=-22.165, z=153.21, rx=-177, ry=-0.095, rz=176.391, fatherId=FrmDraw[0]}
  [594] = {x=-5.103, y=-22.299, z=153.21, rx=-177, ry=-0.138, rz=174.722, fatherId=FrmDraw[0]}
  [595] = {x=-6.714, y=-22.484, z=153.21, rx=-177, ry=-0.182, rz=173.048, fatherId=FrmDraw[0]}
  [596] = {x=-8.325, y=-22.721, z=153.209, rx=-177, ry=-0.226, rz=171.368, fatherId=FrmDraw[0]}
  [597] = {x=-9.934, y=-23.01, z=153.209, rx=-177, ry=-0.271, rz=169.68, fatherId=FrmDraw[0]}
  [598] = {x=-11.543, y=-23.351, z=153.208, rx=-177, ry=-0.316, rz=167.983, fatherId=FrmDraw[0]}
  [599] = {x=-13.15, y=-23.746, z=153.208, rx=-177, ry=-0.361, rz=166.276, fatherId=FrmDraw[0]}
  [600] = {x=-14.756, y=-24.196, z=153.207, rx=-177, ry=-0.407, rz=164.556, fatherId=FrmDraw[0]}
  [601] = {x=-16.361, y=-24.701, z=153.206, rx=-177, ry=-0.453, rz=162.821, fatherId=FrmDraw[0]}
  [602] = {x=-17.964, y=-25.265, z=153.205, rx=-177, ry=-0.5, rz=161.07, fatherId=FrmDraw[0]}
  [603] = {x=-17.983, y=-25.264, z=150.803, rx=-177, ry=-0.5, rz=161.072, fatherId=FrmDraw[0]}
  [604] = {x=-18.004, y=-25.264, z=148.205, rx=-177, ry=-0.5, rz=161.074, fatherId=FrmDraw[0]}
  [605] = {x=-16.397, y=-24.7, z=148.206, rx=-177, ry=-0.453, rz=162.825, fatherId=FrmDraw[0]}
  [606] = {x=-14.789, y=-24.195, z=148.207, rx=-177, ry=-0.407, rz=164.559, fatherId=FrmDraw[0]}
  [607] = {x=-13.179, y=-23.745, z=148.208, rx=-177, ry=-0.361, rz=166.279, fatherId=FrmDraw[0]}
  [608] = {x=-11.568, y=-23.35, z=148.208, rx=-177, ry=-0.316, rz=167.986, fatherId=FrmDraw[0]}
  [609] = {x=-9.956, y=-23.009, z=148.209, rx=-177, ry=-0.271, rz=169.682, fatherId=FrmDraw[0]}
  [610] = {x=-8.343, y=-22.721, z=148.209, rx=-177, ry=-0.226, rz=171.369, fatherId=FrmDraw[0]}
  [611] = {x=-6.729, y=-22.484, z=148.21, rx=-177, ry=-0.182, rz=173.049, fatherId=FrmDraw[0]}
  [612] = {x=-5.115, y=-22.299, z=148.21, rx=-177, ry=-0.138, rz=174.723, fatherId=FrmDraw[0]}
  [613] = {x=-3.5, y=-22.165, z=148.21, rx=-177, ry=-0.095, rz=176.392, fatherId=FrmDraw[0]}
  [614] = {x=-1.885, y=-22.081, z=148.211, rx=-177, ry=-0.051, rz=178.058, fatherId=FrmDraw[0]}
  [615] = {x=-0.808, y=-22.053, z=148.211, rx=-177, ry=-0.022, rz=179.168, fatherId=FrmDraw[0]}
  [616] = {x=0.269, y=-22.048, z=148.211, rx=-177, ry=0.007, rz=-179.723, fatherId=FrmDraw[0]}
  [617] = {x=1.885, y=-22.081, z=148.211, rx=-177, ry=0.051, rz=-178.058, fatherId=FrmDraw[0]}
  [618] = {x=3.5, y=-22.165, z=148.21, rx=-177, ry=0.095, rz=-176.392, fatherId=FrmDraw[0]}
  [619] = {x=5.115, y=-22.299, z=148.21, rx=-177, ry=0.138, rz=-174.723, fatherId=FrmDraw[0]}
  [620] = {x=6.729, y=-22.484, z=148.21, rx=-177, ry=0.182, rz=-173.049, fatherId=FrmDraw[0]}
  [621] = {x=8.343, y=-22.721, z=148.209, rx=-177, ry=0.226, rz=-171.369, fatherId=FrmDraw[0]}
  [622] = {x=9.956, y=-23.009, z=148.209, rx=-177, ry=0.271, rz=-169.682, fatherId=FrmDraw[0]}
  [623] = {x=11.568, y=-23.35, z=148.208, rx=-177, ry=0.316, rz=-167.986, fatherId=FrmDraw[0]}
  [624] = {x=13.179, y=-23.745, z=148.208, rx=-177, ry=0.361, rz=-166.278, fatherId=FrmDraw[0]}
  [625] = {x=14.789, y=-24.195, z=148.207, rx=-177, ry=0.407, rz=-164.559, fatherId=FrmDraw[0]}
  [626] = {x=16.397, y=-24.7, z=148.206, rx=-177, ry=0.453, rz=-162.825, fatherId=FrmDraw[0]}
  [627] = {x=18.004, y=-25.264, z=148.205, rx=-177, ry=0.5, rz=-161.074, fatherId=FrmDraw[0]}
  [628] = {x=18.027, y=-25.264, z=145.803, rx=-177, ry=0.5, rz=-161.072, fatherId=FrmDraw[0]}
  [629] = {x=18.051, y=-25.265, z=143.205, rx=-177, ry=0.5, rz=-161.07, fatherId=FrmDraw[0]}
  [630] = {x=16.44, y=-24.701, z=143.206, rx=-177, ry=0.453, rz=-162.821, fatherId=FrmDraw[0]}
  [631] = {x=14.827, y=-24.196, z=143.207, rx=-177, ry=0.407, rz=-164.556, fatherId=FrmDraw[0]}
  [632] = {x=13.213, y=-23.746, z=143.208, rx=-177, ry=0.361, rz=-166.276, fatherId=FrmDraw[0]}
  [633] = {x=11.598, y=-23.351, z=143.208, rx=-177, ry=0.316, rz=-167.983, fatherId=FrmDraw[0]}
  [634] = {x=9.981, y=-23.009, z=143.209, rx=-177, ry=0.271, rz=-169.68, fatherId=FrmDraw[0]}
  [635] = {x=8.364, y=-22.721, z=143.209, rx=-177, ry=0.226, rz=-171.368, fatherId=FrmDraw[0]}
  [636] = {x=6.746, y=-22.484, z=143.21, rx=-177, ry=0.182, rz=-173.048, fatherId=FrmDraw[0]}
  [637] = {x=5.128, y=-22.299, z=143.21, rx=-177, ry=0.138, rz=-174.722, fatherId=FrmDraw[0]}
  [638] = {x=3.509, y=-22.165, z=143.21, rx=-177, ry=0.095, rz=-176.391, fatherId=FrmDraw[0]}
  [639] = {x=1.889, y=-22.081, z=143.211, rx=-177, ry=0.051, rz=-178.058, fatherId=FrmDraw[0]}
  [640] = {x=0.81, y=-22.053, z=143.211, rx=-177, ry=0.022, rz=-179.168, fatherId=FrmDraw[0]}
  [641] = {x=-0.27, y=-22.048, z=143.211, rx=-177, ry=-0.007, rz=179.723, fatherId=FrmDraw[0]}
  [642] = {x=-1.889, y=-22.081, z=143.211, rx=-177, ry=-0.051, rz=178.058, fatherId=FrmDraw[0]}
  [643] = {x=-3.509, y=-22.165, z=143.21, rx=-177, ry=-0.095, rz=176.391, fatherId=FrmDraw[0]}
  [644] = {x=-5.128, y=-22.299, z=143.21, rx=-177, ry=-0.138, rz=174.722, fatherId=FrmDraw[0]}
  [645] = {x=-6.746, y=-22.484, z=143.21, rx=-177, ry=-0.182, rz=173.048, fatherId=FrmDraw[0]}
  [646] = {x=-8.364, y=-22.721, z=143.209, rx=-177, ry=-0.226, rz=171.368, fatherId=FrmDraw[0]}
  [647] = {x=-9.981, y=-23.01, z=143.209, rx=-177, ry=-0.271, rz=169.68, fatherId=FrmDraw[0]}
  [648] = {x=-11.598, y=-23.351, z=143.208, rx=-177, ry=-0.316, rz=167.983, fatherId=FrmDraw[0]}
  [649] = {x=-13.213, y=-23.746, z=143.208, rx=-177, ry=-0.361, rz=166.276, fatherId=FrmDraw[0]}
  [650] = {x=-14.827, y=-24.196, z=143.207, rx=-177, ry=-0.407, rz=164.556, fatherId=FrmDraw[0]}
  [651] = {x=-16.44, y=-24.701, z=143.206, rx=-177, ry=-0.453, rz=162.821, fatherId=FrmDraw[0]}
  [652] = {x=-18.051, y=-25.265, z=143.205, rx=-177, ry=-0.5, rz=161.071, fatherId=FrmDraw[0]}
  [653] = {x=-18.07, y=-25.264, z=140.803, rx=-177, ry=-0.5, rz=161.072, fatherId=FrmDraw[0]}
  [654] = {x=-18.091, y=-25.264, z=138.205, rx=-177, ry=-0.5, rz=161.074, fatherId=FrmDraw[0]}
  [655] = {x=-16.537, y=-24.72, z=138.206, rx=-177, ry=-0.455, rz=162.76, fatherId=FrmDraw[0]}
  [656] = {x=-15.025, y=-24.244, z=138.207, rx=-177, ry=-0.412, rz=164.383, fatherId=FrmDraw[0]}
  [657] = {x=-13.512, y=-23.816, z=138.208, rx=-177, ry=-0.369, rz=165.993, fatherId=FrmDraw[0]}
  [658] = {x=-11.86, y=-23.405, z=138.208, rx=-177, ry=-0.322, rz=167.737, fatherId=FrmDraw[0]}
  [659] = {x=-10.207, y=-23.049, z=138.209, rx=-177, ry=-0.277, rz=169.469, fatherId=FrmDraw[0]}
  [660] = {x=-8.553, y=-22.749, z=138.209, rx=-177, ry=-0.231, rz=171.192, fatherId=FrmDraw[0]}
  [661] = {x=-6.899, y=-22.502, z=138.21, rx=-177, ry=-0.186, rz=172.906, fatherId=FrmDraw[0]}
  [662] = {x=-5.244, y=-22.31, z=138.21, rx=-177, ry=-0.141, rz=174.615, fatherId=FrmDraw[0]}
  [663] = {x=-3.588, y=-22.17, z=138.21, rx=-177, ry=-0.096, rz=176.318, fatherId=FrmDraw[0]}
  [664] = {x=-1.932, y=-22.082, z=138.211, rx=-177, ry=-0.052, rz=178.018, fatherId=FrmDraw[0]}
  [665] = {x=-0.828, y=-22.053, z=138.211, rx=-177, ry=-0.022, rz=179.151, fatherId=FrmDraw[0]}
  [666] = {x=0.276, y=-22.048, z=138.211, rx=-177, ry=0.007, rz=-179.717, fatherId=FrmDraw[0]}
  [667] = {x=1.932, y=-22.082, z=138.211, rx=-177, ry=0.052, rz=-178.018, fatherId=FrmDraw[0]}
  [668] = {x=3.588, y=-22.17, z=138.21, rx=-177, ry=0.096, rz=-176.318, fatherId=FrmDraw[0]}
  [669] = {x=5.244, y=-22.31, z=138.21, rx=-177, ry=0.141, rz=-174.615, fatherId=FrmDraw[0]}
  [670] = {x=6.899, y=-22.502, z=138.21, rx=-177, ry=0.186, rz=-172.906, fatherId=FrmDraw[0]}
  [671] = {x=8.553, y=-22.749, z=138.209, rx=-177, ry=0.231, rz=-171.192, fatherId=FrmDraw[0]}
  [672] = {x=10.207, y=-23.049, z=138.209, rx=-177, ry=0.277, rz=-169.469, fatherId=FrmDraw[0]}
  [673] = {x=11.86, y=-23.405, z=138.208, rx=-177, ry=0.322, rz=-167.737, fatherId=FrmDraw[0]}
  [674] = {x=13.512, y=-23.816, z=138.208, rx=-177, ry=0.369, rz=-165.993, fatherId=FrmDraw[0]}
  [675] = {x=15.025, y=-24.244, z=138.207, rx=-177, ry=0.412, rz=-164.383, fatherId=FrmDraw[0]}
  [676] = {x=16.537, y=-24.72, z=138.206, rx=-177, ry=0.455, rz=-162.759, fatherId=FrmDraw[0]}
  [677] = {x=18.091, y=-25.264, z=138.205, rx=-177, ry=0.5, rz=-161.074, fatherId=FrmDraw[0]}
  [678] = {x=18.114, y=-25.264, z=135.803, rx=-177, ry=0.5, rz=-161.072, fatherId=FrmDraw[0]}
  [679] = {x=18.138, y=-25.265, z=133.206, rx=-177, ry=0.5, rz=-161.071, fatherId=FrmDraw[0]}
  [680] = {x=16.531, y=-24.705, z=133.206, rx=-177, ry=0.454, rz=-162.809, fatherId=FrmDraw[0]}
  [681] = {x=14.922, y=-24.203, z=133.207, rx=-177, ry=0.408, rz=-164.53, fatherId=FrmDraw[0]}
  [682] = {x=13.312, y=-23.755, z=133.208, rx=-177, ry=0.362, rz=-166.238, fatherId=FrmDraw[0]}
  [683] = {x=11.701, y=-23.362, z=133.209, rx=-177, ry=0.317, rz=-167.933, fatherId=FrmDraw[0]}
  [684] = {x=10.089, y=-23.021, z=133.209, rx=-177, ry=0.273, rz=-169.617, fatherId=FrmDraw[0]}
  [685] = {x=8.476, y=-22.733, z=133.21, rx=-177, ry=0.228, rz=-171.293, fatherId=FrmDraw[0]}
  [686] = {x=6.862, y=-22.495, z=133.21, rx=-177, ry=0.185, rz=-172.961, fatherId=FrmDraw[0]}
  [687] = {x=5.248, y=-22.309, z=133.21, rx=-177, ry=0.141, rz=-174.623, fatherId=FrmDraw[0]}
  [688] = {x=3.634, y=-22.172, z=133.21, rx=-177, ry=0.097, rz=-176.28, fatherId=FrmDraw[0]}
  [689] = {x=2.019, y=-22.086, z=133.211, rx=-177, ry=0.054, rz=-177.934, fatherId=FrmDraw[0]}
  [690] = {x=0.673, y=-22.051, z=133.211, rx=-177, ry=0.018, rz=-179.312, fatherId=FrmDraw[0]}
  [691] = {x=-0.404, y=-22.048, z=133.211, rx=-177, ry=-0.011, rz=179.587, fatherId=FrmDraw[0]}
  [692] = {x=-2.019, y=-22.086, z=133.211, rx=-177, ry=-0.054, rz=177.934, fatherId=FrmDraw[0]}
  [693] = {x=-3.634, y=-22.172, z=133.21, rx=-177, ry=-0.097, rz=176.28, fatherId=FrmDraw[0]}
  [694] = {x=-5.248, y=-22.309, z=133.21, rx=-177, ry=-0.141, rz=174.623, fatherId=FrmDraw[0]}
  [695] = {x=-6.862, y=-22.495, z=133.21, rx=-177, ry=-0.185, rz=172.961, fatherId=FrmDraw[0]}
  [696] = {x=-8.476, y=-22.733, z=133.21, rx=-177, ry=-0.228, rz=171.293, fatherId=FrmDraw[0]}
  [697] = {x=-10.089, y=-23.021, z=133.209, rx=-177, ry=-0.273, rz=169.617, fatherId=FrmDraw[0]}
  [698] = {x=-11.701, y=-23.362, z=133.209, rx=-177, ry=-0.317, rz=167.933, fatherId=FrmDraw[0]}
  [699] = {x=-13.312, y=-23.755, z=133.208, rx=-177, ry=-0.362, rz=166.238, fatherId=FrmDraw[0]}
  [700] = {x=-14.922, y=-24.203, z=133.207, rx=-177, ry=-0.408, rz=164.53, fatherId=FrmDraw[0]}
  [701] = {x=-16.531, y=-24.705, z=133.206, rx=-177, ry=-0.454, rz=162.809, fatherId=FrmDraw[0]}
  [702] = {x=-18.138, y=-25.265, z=133.206, rx=-177, ry=-0.5, rz=161.071, fatherId=FrmDraw[0]}
  [703] = {x=-18.162, y=-25.265, z=130.659, rx=-177, ry=-0.5, rz=161.069, fatherId=FrmDraw[0]}
  [704] = {x=-16.552, y=-24.706, z=130.66, rx=-177, ry=-0.454, rz=162.808, fatherId=FrmDraw[0]}
  [705] = {x=-14.941, y=-24.203, z=130.661, rx=-177, ry=-0.408, rz=164.529, fatherId=FrmDraw[0]}
  [706] = {x=-13.329, y=-23.755, z=130.662, rx=-177, ry=-0.362, rz=166.237, fatherId=FrmDraw[0]}
  [707] = {x=-11.716, y=-23.362, z=130.662, rx=-177, ry=-0.317, rz=167.932, fatherId=FrmDraw[0]}
  [708] = {x=-10.102, y=-23.021, z=130.663, rx=-177, ry=-0.273, rz=169.617, fatherId=FrmDraw[0]}
  [709] = {x=-8.487, y=-22.733, z=130.663, rx=-177, ry=-0.228, rz=171.292, fatherId=FrmDraw[0]}
  [710] = {x=-6.871, y=-22.495, z=130.663, rx=-177, ry=-0.185, rz=172.96, fatherId=FrmDraw[0]}
  [711] = {x=-5.255, y=-22.309, z=130.664, rx=-177, ry=-0.141, rz=174.622, fatherId=FrmDraw[0]}
  [712] = {x=-3.638, y=-22.172, z=130.664, rx=-177, ry=-0.097, rz=176.28, fatherId=FrmDraw[0]}
  [713] = {x=-2.021, y=-22.086, z=130.664, rx=-177, ry=-0.054, rz=177.934, fatherId=FrmDraw[0]}
  [714] = {x=-0.674, y=-22.051, z=130.664, rx=-177, ry=-0.018, rz=179.312, fatherId=FrmDraw[0]}
  [715] = {x=0.404, y=-22.048, z=130.664, rx=-177, ry=0.011, rz=-179.587, fatherId=FrmDraw[0]}
  [716] = {x=2.021, y=-22.086, z=130.664, rx=-177, ry=0.054, rz=-177.934, fatherId=FrmDraw[0]}
  [717] = {x=3.638, y=-22.172, z=130.664, rx=-177, ry=0.097, rz=-176.28, fatherId=FrmDraw[0]}
  [718] = {x=5.255, y=-22.309, z=130.664, rx=-177, ry=0.141, rz=-174.622, fatherId=FrmDraw[0]}
  [719] = {x=6.871, y=-22.495, z=130.663, rx=-177, ry=0.185, rz=-172.96, fatherId=FrmDraw[0]}
  [720] = {x=8.487, y=-22.733, z=130.663, rx=-177, ry=0.228, rz=-171.292, fatherId=FrmDraw[0]}
  [721] = {x=10.102, y=-23.021, z=130.663, rx=-177, ry=0.273, rz=-169.617, fatherId=FrmDraw[0]}
  [722] = {x=11.716, y=-23.362, z=130.662, rx=-177, ry=0.317, rz=-167.932, fatherId=FrmDraw[0]}
  [723] = {x=13.329, y=-23.755, z=130.662, rx=-177, ry=0.362, rz=-166.237, fatherId=FrmDraw[0]}
  [724] = {x=14.941, y=-24.203, z=130.661, rx=-177, ry=0.408, rz=-164.529, fatherId=FrmDraw[0]}
  [725] = {x=16.552, y=-24.706, z=130.66, rx=-177, ry=0.454, rz=-162.807, fatherId=FrmDraw[0]}
  [726] = {x=18.162, y=-25.265, z=130.659, rx=-177, ry=0.5, rz=-161.069, fatherId=FrmDraw[0]}
  [727] = {x=18.185, y=-25.266, z=128.087, rx=-177, ry=0.5, rz=-161.069, fatherId=FrmDraw[0]}
  [728] = {x=16.573, y=-24.706, z=128.088, rx=-177, ry=0.454, rz=-162.807, fatherId=FrmDraw[0]}
  [729] = {x=14.96, y=-24.203, z=128.089, rx=-177, ry=0.408, rz=-164.529, fatherId=FrmDraw[0]}
  [730] = {x=13.346, y=-23.755, z=128.09, rx=-177, ry=0.362, rz=-166.236, fatherId=FrmDraw[0]}
  [731] = {x=11.731, y=-23.362, z=128.09, rx=-177, ry=0.317, rz=-167.932, fatherId=FrmDraw[0]}
  [732] = {x=10.114, y=-23.021, z=128.091, rx=-177, ry=0.273, rz=-169.616, fatherId=FrmDraw[0]}
  [733] = {x=8.497, y=-22.733, z=128.091, rx=-177, ry=0.228, rz=-171.292, fatherId=FrmDraw[0]}
  [734] = {x=6.88, y=-22.495, z=128.092, rx=-177, ry=0.185, rz=-172.96, fatherId=FrmDraw[0]}
  [735] = {x=5.261, y=-22.309, z=128.092, rx=-177, ry=0.141, rz=-174.622, fatherId=FrmDraw[0]}
  [736] = {x=3.643, y=-22.172, z=128.092, rx=-177, ry=0.097, rz=-176.28, fatherId=FrmDraw[0]}
  [737] = {x=2.024, y=-22.086, z=128.092, rx=-177, ry=0.054, rz=-177.934, fatherId=FrmDraw[0]}
  [738] = {x=0.675, y=-22.051, z=128.092, rx=-177, ry=0.018, rz=-179.312, fatherId=FrmDraw[0]}
  [739] = {x=-0.405, y=-22.048, z=128.092, rx=-177, ry=-0.011, rz=179.587, fatherId=FrmDraw[0]}
  [740] = {x=-2.024, y=-22.086, z=128.092, rx=-177, ry=-0.054, rz=177.934, fatherId=FrmDraw[0]}
  [741] = {x=-3.643, y=-22.172, z=128.092, rx=-177, ry=-0.097, rz=176.28, fatherId=FrmDraw[0]}
  [742] = {x=-5.261, y=-22.309, z=128.092, rx=-177, ry=-0.141, rz=174.622, fatherId=FrmDraw[0]}
  [743] = {x=-6.879, y=-22.496, z=128.092, rx=-177, ry=-0.185, rz=172.96, fatherId=FrmDraw[0]}
  [744] = {x=-8.497, y=-22.733, z=128.091, rx=-177, ry=-0.228, rz=171.292, fatherId=FrmDraw[0]}
  [745] = {x=-10.114, y=-23.021, z=128.091, rx=-177, ry=-0.273, rz=169.616, fatherId=FrmDraw[0]}
  [746] = {x=-11.731, y=-23.362, z=128.09, rx=-177, ry=-0.317, rz=167.932, fatherId=FrmDraw[0]}
  [747] = {x=-13.346, y=-23.755, z=128.09, rx=-177, ry=-0.362, rz=166.236, fatherId=FrmDraw[0]}
  [748] = {x=-14.96, y=-24.203, z=128.089, rx=-177, ry=-0.408, rz=164.529, fatherId=FrmDraw[0]}
  [749] = {x=-16.573, y=-24.706, z=128.088, rx=-177, ry=-0.454, rz=162.807, fatherId=FrmDraw[0]}
  [750] = {x=-18.185, y=-25.266, z=128.087, rx=-177, ry=-0.5, rz=161.069, fatherId=FrmDraw[0]}
  [751] = {x=-18.208, y=-25.266, z=125.49, rx=-177, ry=-0.5, rz=161.068, fatherId=FrmDraw[0]}
  [752] = {x=-16.594, y=-24.706, z=125.491, rx=-177, ry=-0.454, rz=162.806, fatherId=FrmDraw[0]}
  [753] = {x=-14.979, y=-24.203, z=125.491, rx=-177, ry=-0.408, rz=164.528, fatherId=FrmDraw[0]}
  [754] = {x=-13.363, y=-23.756, z=125.492, rx=-177, ry=-0.362, rz=166.236, fatherId=FrmDraw[0]}
  [755] = {x=-11.745, y=-23.362, z=125.493, rx=-177, ry=-0.317, rz=167.932, fatherId=FrmDraw[0]}
  [756] = {x=-10.127, y=-23.021, z=125.493, rx=-177, ry=-0.273, rz=169.616, fatherId=FrmDraw[0]}
  [757] = {x=-8.508, y=-22.733, z=125.494, rx=-177, ry=-0.228, rz=171.292, fatherId=FrmDraw[0]}
  [758] = {x=-6.888, y=-22.496, z=125.494, rx=-177, ry=-0.185, rz=172.96, fatherId=FrmDraw[0]}
  [759] = {x=-5.268, y=-22.309, z=125.494, rx=-177, ry=-0.141, rz=174.622, fatherId=FrmDraw[0]}
  [760] = {x=-3.647, y=-22.172, z=125.494, rx=-177, ry=-0.097, rz=176.28, fatherId=FrmDraw[0]}
  [761] = {x=-2.026, y=-22.086, z=125.495, rx=-177, ry=-0.054, rz=177.934, fatherId=FrmDraw[0]}
  [762] = {x=-0.675, y=-22.051, z=125.495, rx=-177, ry=-0.018, rz=179.312, fatherId=FrmDraw[0]}
  [763] = {x=0.405, y=-22.048, z=125.495, rx=-177, ry=0.011, rz=-179.587, fatherId=FrmDraw[0]}
  [764] = {x=2.026, y=-22.086, z=125.495, rx=-177, ry=0.054, rz=-177.934, fatherId=FrmDraw[0]}
  [765] = {x=3.647, y=-22.172, z=125.494, rx=-177, ry=0.097, rz=-176.28, fatherId=FrmDraw[0]}
  [766] = {x=5.268, y=-22.309, z=125.494, rx=-177, ry=0.141, rz=-174.622, fatherId=FrmDraw[0]}
  [767] = {x=6.888, y=-22.496, z=125.494, rx=-177, ry=0.185, rz=-172.96, fatherId=FrmDraw[0]}
  [768] = {x=8.508, y=-22.733, z=125.494, rx=-177, ry=0.228, rz=-171.292, fatherId=FrmDraw[0]}
  [769] = {x=10.127, y=-23.021, z=125.493, rx=-177, ry=0.273, rz=-169.616, fatherId=FrmDraw[0]}
  [770] = {x=11.745, y=-23.362, z=125.493, rx=-177, ry=0.317, rz=-167.931, fatherId=FrmDraw[0]}
  [771] = {x=13.363, y=-23.756, z=125.492, rx=-177, ry=0.362, rz=-166.236, fatherId=FrmDraw[0]}
  [772] = {x=14.979, y=-24.203, z=125.491, rx=-177, ry=0.408, rz=-164.528, fatherId=FrmDraw[0]}
  [773] = {x=16.594, y=-24.706, z=125.491, rx=-177, ry=0.454, rz=-162.806, fatherId=FrmDraw[0]}
  [774] = {x=18.208, y=-25.266, z=125.49, rx=-177, ry=0.5, rz=-161.068, fatherId=FrmDraw[0]}
  [775] = {x=18.225, y=-25.264, z=123.02, rx=-177, ry=0.5, rz=-161.073, fatherId=FrmDraw[0]}
  [776] = {x=16.61, y=-24.705, z=123.021, rx=-177, ry=0.454, rz=-162.811, fatherId=FrmDraw[0]}
  [777] = {x=14.993, y=-24.202, z=123.022, rx=-177, ry=0.408, rz=-164.532, fatherId=FrmDraw[0]}
  [778] = {x=13.375, y=-23.755, z=123.022, rx=-177, ry=0.362, rz=-166.24, fatherId=FrmDraw[0]}
  [779] = {x=11.756, y=-23.361, z=123.023, rx=-177, ry=0.317, rz=-167.935, fatherId=FrmDraw[0]}
  [780] = {x=10.136, y=-23.021, z=123.023, rx=-177, ry=0.273, rz=-169.619, fatherId=FrmDraw[0]}
  [781] = {x=8.515, y=-22.732, z=123.024, rx=-177, ry=0.228, rz=-171.294, fatherId=FrmDraw[0]}
  [782] = {x=6.894, y=-22.495, z=123.024, rx=-177, ry=0.185, rz=-172.962, fatherId=FrmDraw[0]}
  [783] = {x=5.273, y=-22.309, z=123.024, rx=-177, ry=0.141, rz=-174.623, fatherId=FrmDraw[0]}
  [784] = {x=3.65, y=-22.172, z=123.025, rx=-177, ry=0.097, rz=-176.281, fatherId=FrmDraw[0]}
  [785] = {x=2.028, y=-22.086, z=123.025, rx=-177, ry=0.054, rz=-177.935, fatherId=FrmDraw[0]}
  [786] = {x=0.676, y=-22.051, z=123.025, rx=-177, ry=0.018, rz=-179.312, fatherId=FrmDraw[0]}
  [787] = {x=-0.406, y=-22.048, z=123.025, rx=-177, ry=-0.011, rz=179.587, fatherId=FrmDraw[0]}
  [788] = {x=-2.028, y=-22.086, z=123.025, rx=-177, ry=-0.054, rz=177.935, fatherId=FrmDraw[0]}
  [789] = {x=-3.65, y=-22.172, z=123.025, rx=-177, ry=-0.097, rz=176.281, fatherId=FrmDraw[0]}
  [790] = {x=-5.273, y=-22.309, z=123.024, rx=-177, ry=-0.141, rz=174.623, fatherId=FrmDraw[0]}
  [791] = {x=-6.894, y=-22.495, z=123.024, rx=-177, ry=-0.185, rz=172.962, fatherId=FrmDraw[0]}
  [792] = {x=-8.515, y=-22.732, z=123.024, rx=-177, ry=-0.228, rz=171.294, fatherId=FrmDraw[0]}
  [793] = {x=-10.136, y=-23.021, z=123.023, rx=-177, ry=-0.273, rz=169.619, fatherId=FrmDraw[0]}
  [794] = {x=-11.756, y=-23.361, z=123.023, rx=-177, ry=-0.317, rz=167.935, fatherId=FrmDraw[0]}
  [795] = {x=-13.375, y=-23.755, z=123.022, rx=-177, ry=-0.362, rz=166.24, fatherId=FrmDraw[0]}
  [796] = {x=-14.993, y=-24.202, z=123.022, rx=-177, ry=-0.408, rz=164.533, fatherId=FrmDraw[0]}
  [797] = {x=-16.61, y=-24.705, z=123.021, rx=-177, ry=-0.454, rz=162.811, fatherId=FrmDraw[0]}
  [798] = {x=-18.225, y=-25.264, z=123.02, rx=-177, ry=-0.5, rz=161.073, fatherId=FrmDraw[0]}
public pointRx shere = {x=16.915, y=-25.265, z=273.2, rx=-177, ry=0.5, rz=-161.069, fatherId=FrmDraw[0]}
string sString[1500]
  [0] = "16.915000,-25.265000,273.200000,-177.000000,0.500000,-161.069000,"
  [1] = "15.593000,-24.767000,273.202000,-177.000000,0.459000,-162.610000,"
  [2] = "14.003000,-24.227000,273.204000,-177.000000,0.410000,-164.442000,"
  [3] = "12.409000,-23.750000,273.205000,-177.000000,0.362000,-166.257000,"
  [4] = "10.813000,-23.335000,273.207000,-177.000000,0.314000,-168.059000,"
  [5] = "9.215000,-22.978000,273.208000,-177.000000,0.267000,-169.848000,"
  [6] = "7.615000,-22.681000,273.209000,-177.000000,0.220000,-171.628000,"
  [7] = "6.014000,-22.441000,273.209000,-177.000000,0.173000,-173.399000,"
  [8] = "4.411000,-22.259000,273.210000,-177.000000,0.127000,-175.164000,"
  [9] = "2.807000,-22.133000,273.210000,-177.000000,0.081000,-176.925000,"
  [10] = "1.203000,-22.063000,273.211000,-177.000000,0.034000,-178.683000,"
  [11] = "0.134000,-22.047000,273.211000,-177.000000,0.004000,-179.854000,"
  [12] = "-1.203000,-22.063000,273.211000,-177.000000,-0.034000,178.683000,"
  [13] = "-2.807000,-22.133000,273.210000,-177.000000,-0.081000,176.925000,"
  [14] = "-4.411000,-22.259000,273.210000,-177.000000,-0.127000,175.164000,"
  [15] = "-6.014000,-22.441000,273.209000,-177.000000,-0.173000,173.399000,"
  [16] = "-7.615000,-22.681000,273.209000,-177.000000,-0.220000,171.628000,"
  [17] = "-9.215000,-22.978000,273.208000,-177.000000,-0.267000,169.848000,"
  [18] = "-10.813000,-23.335000,273.207000,-177.000000,-0.314000,168.059000,"
  [19] = "-12.409000,-23.750000,273.205000,-177.000000,-0.362000,166.257000,"
  [20] = "-14.002000,-24.227000,273.204000,-177.000000,-0.410000,164.442000,"
  [21] = "-15.593000,-24.767000,273.202000,-177.000000,-0.459000,162.610000,"
  [22] = "-16.915000,-25.265000,273.200000,-177.000000,-0.500000,161.069000,"
  [23] = "-16.935000,-25.265000,270.798000,-177.000000,-0.500000,161.071000,"
  [24] = "-16.956000,-25.264000,268.200000,-177.000000,-0.500000,161.073000,"
  [25] = "-15.630000,-24.766000,268.202000,-177.000000,-0.459000,162.614000,"
  [26] = "-14.035000,-24.226000,268.204000,-177.000000,-0.410000,164.445000,"
  [27] = "-12.438000,-23.750000,268.205000,-177.000000,-0.362000,166.260000,"
  [28] = "-10.838000,-23.334000,268.207000,-177.000000,-0.314000,168.061000,"
  [29] = "-9.236000,-22.978000,268.208000,-177.000000,-0.266000,169.850000,"
  [30] = "-7.633000,-22.681000,268.209000,-177.000000,-0.220000,171.630000,"
  [31] = "-6.027000,-22.441000,268.209000,-177.000000,-0.173000,173.401000,"
  [32] = "-4.421000,-22.259000,268.210000,-177.000000,-0.127000,175.165000,"
  [33] = "-2.814000,-22.133000,268.210000,-177.000000,-0.081000,176.926000,"
  [34] = "-1.206000,-22.063000,268.211000,-177.000000,-0.034000,178.683000,"
  [35] = "-0.134000,-22.047000,268.211000,-177.000000,-0.004000,179.854000,"
  [36] = "1.206000,-22.063000,268.211000,-177.000000,0.034000,-178.683000,"
  [37] = "2.814000,-22.133000,268.210000,-177.000000,0.081000,-176.926000,"
  [38] = "4.421000,-22.259000,268.210000,-177.000000,0.127000,-175.165000,"
  [39] = "6.027000,-22.441000,268.209000,-177.000000,0.173000,-173.401000,"
  [40] = "7.633000,-22.681000,268.209000,-177.000000,0.220000,-171.630000,"
  [41] = "9.237000,-22.978000,268.208000,-177.000000,0.266000,-169.850000,"
  [42] = "10.838000,-23.334000,268.207000,-177.000000,0.314000,-168.061000,"
  [43] = "12.438000,-23.750000,268.205000,-177.000000,0.362000,-166.260000,"
  [44] = "14.035000,-24.226000,268.204000,-177.000000,0.410000,-164.445000,"
  [45] = "15.630000,-24.766000,268.202000,-177.000000,0.459000,-162.614000,"
  [46] = "16.956000,-25.264000,268.200000,-177.000000,0.500000,-161.073000,"
  [47] = "16.978000,-25.265000,265.798000,-177.000000,0.500000,-161.071000,"
  [48] = "17.003000,-25.265000,263.201000,-177.000000,0.500000,-161.069000,"
  [49] = "15.673000,-24.767000,263.202000,-177.000000,0.459000,-162.610000,"
  [50] = "14.074000,-24.227000,263.204000,-177.000000,0.410000,-164.442000,"
  [51] = "12.472000,-23.750000,263.205000,-177.000000,0.362000,-166.257000,"
  [52] = "10.868000,-23.335000,263.207000,-177.000000,0.314000,-168.059000,"
  [53] = "9.262000,-22.978000,263.208000,-177.000000,0.267000,-169.848000,"
  [54] = "7.653000,-22.681000,263.209000,-177.000000,0.220000,-171.628000,"
  [55] = "6.044000,-22.441000,263.209000,-177.000000,0.173000,-173.399000,"
  [56] = "4.433000,-22.259000,263.210000,-177.000000,0.127000,-175.164000,"
  [57] = "2.821000,-22.133000,263.210000,-177.000000,0.081000,-176.925000,"
  [58] = "1.209000,-22.063000,263.211000,-177.000000,0.034000,-178.683000,"
  [59] = "0.134000,-22.047000,263.211000,-177.000000,0.004000,-179.854000,"
  [60] = "-1.209000,-22.063000,263.211000,-177.000000,-0.034000,178.683000,"
  [61] = "-2.821000,-22.133000,263.210000,-177.000000,-0.081000,176.925000,"
  [62] = "-4.433000,-22.259000,263.210000,-177.000000,-0.127000,175.165000,"
  [63] = "-6.044000,-22.441000,263.209000,-177.000000,-0.173000,173.399000,"
  [64] = "-7.653000,-22.681000,263.209000,-177.000000,-0.220000,171.628000,"
  [65] = "-9.262000,-22.978000,263.208000,-177.000000,-0.267000,169.848000,"
  [66] = "-10.868000,-23.335000,263.207000,-177.000000,-0.314000,168.059000,"
  [67] = "-12.472000,-23.750000,263.205000,-177.000000,-0.362000,166.257000,"
  [68] = "-14.074000,-24.227000,263.204000,-177.000000,-0.410000,164.442000,"
  [69] = "-15.673000,-24.767000,263.202000,-177.000000,-0.459000,162.610000,"
  [70] = "-17.003000,-25.265000,263.201000,-177.000000,-0.500000,161.069000,"
  [71] = "-17.022000,-25.265000,260.799000,-177.000000,-0.500000,161.071000,"
  [72] = "-17.043000,-25.264000,258.201000,-177.000000,-0.500000,161.074000,"
  [73] = "-15.455000,-24.676000,258.203000,-177.000000,-0.451000,162.906000,"
  [74] = "-13.865000,-24.150000,258.204000,-177.000000,-0.403000,164.720000,"
  [75] = "-12.271000,-23.686000,258.206000,-177.000000,-0.355000,166.519000,"
  [76] = "-10.675000,-23.282000,258.207000,-177.000000,-0.307000,168.304000,"
  [77] = "-9.077000,-22.937000,258.208000,-177.000000,-0.260000,170.078000,"
  [78] = "-7.478000,-22.649000,258.209000,-177.000000,-0.214000,171.842000,"
  [79] = "-5.877000,-22.418000,258.209000,-177.000000,-0.168000,173.599000,"
  [80] = "-4.275000,-22.243000,258.210000,-177.000000,-0.122000,175.349000,"
  [81] = "-2.672000,-22.123000,258.210000,-177.000000,-0.076000,177.095000,"
  [82] = "-1.069000,-22.059000,258.211000,-177.000000,-0.030000,178.838000,"
  [83] = "0.000000,-22.047000,258.211000,-177.000000,0.000000,180.000000,"
  [84] = "1.069000,-22.059000,258.211000,-177.000000,0.030000,-178.838000,"
  [85] = "2.672000,-22.123000,258.210000,-177.000000,0.076000,-177.095000,"
  [86] = "4.275000,-22.243000,258.210000,-177.000000,0.122000,-175.349000,"
  [87] = "5.877000,-22.418000,258.209000,-177.000000,0.168000,-173.599000,"
  [88] = "7.478000,-22.649000,258.209000,-177.000000,0.214000,-171.842000,"
  [89] = "9.077000,-22.937000,258.208000,-177.000000,0.260000,-170.078000,"
  [90] = "10.675000,-23.282000,258.207000,-177.000000,0.307000,-168.304000,"
  [91] = "12.271000,-23.686000,258.206000,-177.000000,0.355000,-166.519000,"
  [92] = "13.865000,-24.150000,258.204000,-177.000000,0.403000,-164.720000,"
  [93] = "15.455000,-24.676000,258.203000,-177.000000,0.451000,-162.906000,"
  [94] = "17.043000,-25.264000,258.201000,-177.000000,0.500000,-161.073000,"
  [95] = "17.066000,-25.265000,255.799000,-177.000000,0.500000,-161.072000,"
  [96] = "17.090000,-25.265000,253.201000,-177.000000,0.500000,-161.070000,"
  [97] = "15.763000,-24.770000,253.203000,-177.000000,0.459000,-162.598000,"
  [98] = "14.169000,-24.234000,253.204000,-177.000000,0.411000,-164.416000,"
  [99] = "12.571000,-23.760000,253.206000,-177.000000,0.363000,-166.217000,"
  [100] = "10.971000,-23.346000,253.207000,-177.000000,0.315000,-168.005000,"
  [101] = "9.369000,-22.991000,253.208000,-177.000000,0.268000,-169.781000,"
  [102] = "7.765000,-22.693000,253.209000,-177.000000,0.222000,-171.547000,"
  [103] = "6.160000,-22.453000,253.209000,-177.000000,0.176000,-173.305000,"
  [104] = "4.554000,-22.268000,253.210000,-177.000000,0.130000,-175.057000,"
  [105] = "2.947000,-22.139000,253.210000,-177.000000,0.084000,-176.804000,"
  [106] = "1.340000,-22.066000,253.211000,-177.000000,0.038000,-178.548000,"
  [107] = "0.268000,-22.048000,253.211000,-177.000000,0.008000,-179.710000,"
  [108] = "-1.340000,-22.066000,253.211000,-177.000000,-0.038000,178.548000,"
  [109] = "-2.947000,-22.139000,253.210000,-177.000000,-0.084000,176.804000,"
  [110] = "-4.554000,-22.268000,253.210000,-177.000000,-0.130000,175.057000,"
  [111] = "-6.160000,-22.453000,253.209000,-177.000000,-0.176000,173.305000,"
  [112] = "-7.765000,-22.693000,253.209000,-177.000000,-0.222000,171.547000,"
  [113] = "-9.369000,-22.991000,253.208000,-177.000000,-0.268000,169.781000,"
  [114] = "-10.971000,-23.346000,253.207000,-177.000000,-0.315000,168.005000,"
  [115] = "-12.571000,-23.760000,253.206000,-177.000000,-0.363000,166.217000,"
  [116] = "-14.169000,-24.234000,253.204000,-177.000000,-0.411000,164.416000,"
  [117] = "-15.763000,-24.770000,253.203000,-177.000000,-0.459000,162.598000,"
  [118] = "-17.090000,-25.265000,253.201000,-177.000000,-0.500000,161.070000,"
  [119] = "-17.109000,-25.265000,250.799000,-177.000000,-0.500000,161.071000,"
  [120] = "-17.130000,-25.264000,248.201000,-177.000000,-0.500000,161.074000,"
  [121] = "-15.800000,-24.769000,248.203000,-177.000000,-0.459000,162.602000,"
  [122] = "-14.202000,-24.234000,248.204000,-177.000000,-0.411000,164.419000,"
  [123] = "-12.600000,-23.760000,248.206000,-177.000000,-0.363000,166.220000,"
  [124] = "-10.996000,-23.346000,248.207000,-177.000000,-0.315000,168.007000,"
  [125] = "-9.391000,-22.990000,248.208000,-177.000000,-0.268000,169.783000,"
  [126] = "-7.783000,-22.693000,248.209000,-177.000000,-0.222000,171.549000,"
  [127] = "-6.174000,-22.453000,248.209000,-177.000000,-0.175000,173.306000,"
  [128] = "-4.565000,-22.268000,248.210000,-177.000000,-0.130000,175.058000,"
  [129] = "-2.954000,-22.139000,248.210000,-177.000000,-0.084000,176.804000,"
  [130] = "-1.343000,-22.066000,248.211000,-177.000000,-0.038000,178.548000,"
  [131] = "0.000000,-22.047000,248.211000,-177.000000,0.000000,180.000000,"
  [132] = "1.343000,-22.066000,248.211000,-177.000000,0.038000,-178.548000,"
  [133] = "2.954000,-22.139000,248.210000,-177.000000,0.084000,-176.804000,"
  [134] = "4.565000,-22.268000,248.210000,-177.000000,0.130000,-175.058000,"
  [135] = "6.174000,-22.453000,248.209000,-177.000000,0.175000,-173.306000,"
  [136] = "7.783000,-22.693000,248.209000,-177.000000,0.222000,-171.549000,"
  [137] = "9.391000,-22.990000,248.208000,-177.000000,0.268000,-169.783000,"
  [138] = "10.997000,-23.346000,248.207000,-177.000000,0.315000,-168.007000,"
  [139] = "12.600000,-23.760000,248.206000,-177.000000,0.363000,-166.220000,"
  [140] = "14.202000,-24.234000,248.204000,-177.000000,0.411000,-164.419000,"
  [141] = "15.800000,-24.769000,248.203000,-177.000000,0.459000,-162.602000,"
  [142] = "17.130000,-25.264000,248.201000,-177.000000,0.500000,-161.074000,"
  [143] = "17.153000,-25.265000,245.799000,-177.000000,0.500000,-161.072000,"
  [144] = "17.177000,-25.265000,243.201000,-177.000000,0.500000,-161.070000,"
  [145] = "15.589000,-24.681000,243.203000,-177.000000,0.451000,-162.888000,"
  [146] = "13.998000,-24.159000,243.205000,-177.000000,0.403000,-164.689000,"
  [147] = "12.404000,-23.697000,243.206000,-177.000000,0.356000,-166.474000,"
  [148] = "10.808000,-23.294000,243.207000,-177.000000,0.309000,-168.247000,"
  [149] = "9.210000,-22.950000,243.208000,-177.000000,0.262000,-170.007000,"
  [150] = "7.610000,-22.661000,243.209000,-177.000000,0.216000,-171.759000,"
  [151] = "6.010000,-22.429000,243.210000,-177.000000,0.170000,-173.502000,"
  [152] = "4.408000,-22.252000,243.210000,-177.000000,0.125000,-175.240000,"
  [153] = "2.805000,-22.130000,243.210000,-177.000000,0.079000,-176.973000,"
  [154] = "1.202000,-22.062000,243.211000,-177.000000,0.034000,-178.703000,"
  [155] = "0.134000,-22.047000,243.211000,-177.000000,0.004000,-179.856000,"
  [156] = "-1.202000,-22.062000,243.211000,-177.000000,-0.034000,178.703000,"
  [157] = "-2.805000,-22.130000,243.210000,-177.000000,-0.079000,176.973000,"
  [158] = "-4.408000,-22.252000,243.210000,-177.000000,-0.125000,175.240000,"
  [159] = "-6.010000,-22.429000,243.210000,-177.000000,-0.170000,173.502000,"
  [160] = "-7.610000,-22.661000,243.209000,-177.000000,-0.216000,171.759000,"
  [161] = "-9.210000,-22.950000,243.208000,-177.000000,-0.262000,170.007000,"
  [162] = "-10.808000,-23.294000,243.207000,-177.000000,-0.309000,168.247000,"
  [163] = "-12.404000,-23.697000,243.206000,-177.000000,-0.356000,166.474000,"
  [164] = "-13.998000,-24.159000,243.205000,-177.000000,-0.403000,164.689000,"
  [165] = "-15.589000,-24.681000,243.203000,-177.000000,-0.451000,162.888000,"
  [166] = "-17.177000,-25.265000,243.201000,-177.000000,-0.500000,161.070000,"
  [167] = "-17.197000,-25.265000,240.799000,-177.000000,-0.500000,161.072000,"
  [168] = "-17.218000,-25.264000,238.202000,-177.000000,-0.500000,161.074000,"
  [169] = "-15.625000,-24.680000,238.203000,-177.000000,-0.451000,162.892000,"
  [170] = "-14.030000,-24.158000,238.205000,-177.000000,-0.403000,164.692000,"
  [171] = "-12.433000,-23.696000,238.206000,-177.000000,-0.356000,166.477000,"
  [172] = "-10.833000,-23.294000,238.207000,-177.000000,-0.309000,168.249000,"
  [173] = "-9.231000,-22.949000,238.208000,-177.000000,-0.262000,170.009000,"
  [174] = "-7.628000,-22.661000,238.209000,-177.000000,-0.216000,171.760000,"
  [175] = "-6.023000,-22.429000,238.210000,-177.000000,-0.170000,173.503000,"
  [176] = "-4.418000,-22.252000,238.210000,-177.000000,-0.125000,175.241000,"
  [177] = "-2.812000,-22.130000,238.210000,-177.000000,-0.079000,176.973000,"
  [178] = "-1.205000,-22.062000,238.211000,-177.000000,-0.034000,178.703000,"
  [179] = "-0.134000,-22.047000,238.211000,-177.000000,-0.004000,179.856000,"
  [180] = "1.205000,-22.062000,238.211000,-177.000000,0.034000,-178.703000,"
  [181] = "2.812000,-22.130000,238.210000,-177.000000,0.079000,-176.973000,"
  [182] = "4.418000,-22.252000,238.210000,-177.000000,0.125000,-175.241000,"
  [183] = "6.023000,-22.429000,238.210000,-177.000000,0.170000,-173.503000,"
  [184] = "7.628000,-22.661000,238.209000,-177.000000,0.216000,-171.760000,"
  [185] = "9.231000,-22.949000,238.208000,-177.000000,0.262000,-170.009000,"
  [186] = "10.833000,-23.294000,238.207000,-177.000000,0.309000,-168.249000,"
  [187] = "12.433000,-23.697000,238.206000,-177.000000,0.356000,-166.477000,"
  [188] = "14.030000,-24.158000,238.205000,-177.000000,0.403000,-164.692000,"
  [189] = "15.625000,-24.680000,238.203000,-177.000000,0.451000,-162.892000,"
  [190] = "17.218000,-25.264000,238.202000,-177.000000,0.500000,-161.074000,"
  [191] = "17.240000,-25.265000,235.800000,-177.000000,0.500000,-161.072000,"
  [192] = "17.265000,-25.265000,233.202000,-177.000000,0.500000,-161.070000,"
  [193] = "15.934000,-24.774000,233.203000,-177.000000,0.460000,-162.586000,"
  [194] = "14.335000,-24.242000,233.205000,-177.000000,0.411000,-164.390000,"
  [195] = "12.733000,-23.770000,233.206000,-177.000000,0.364000,-166.178000,"
  [196] = "11.129000,-23.358000,233.207000,-177.000000,0.317000,-167.952000,"
  [197] = "9.524000,-23.003000,233.208000,-177.000000,0.270000,-169.715000,"
  [198] = "7.916000,-22.706000,233.209000,-177.000000,0.224000,-171.467000,"
  [199] = "6.308000,-22.464000,233.209000,-177.000000,0.178000,-173.212000,"
  [200] = "4.698000,-22.278000,233.210000,-177.000000,0.132000,-174.950000,"
  [201] = "3.088000,-22.147000,233.210000,-177.000000,0.087000,-176.684000,"
  [202] = "1.477000,-22.070000,233.211000,-177.000000,0.042000,-178.415000,"
  [203] = "0.134000,-22.047000,233.211000,-177.000000,0.004000,-179.856000,"
  [204] = "-1.477000,-22.070000,233.211000,-177.000000,-0.042000,178.415000,"
  [205] = "-3.088000,-22.147000,233.210000,-177.000000,-0.087000,176.684000,"
  [206] = "-4.698000,-22.278000,233.210000,-177.000000,-0.132000,174.950000,"
  [207] = "-6.308000,-22.464000,233.209000,-177.000000,-0.178000,173.212000,"
  [208] = "-7.916000,-22.706000,233.209000,-177.000000,-0.224000,171.467000,"
  [209] = "-9.524000,-23.003000,233.208000,-177.000000,-0.270000,169.715000,"
  [210] = "-11.129000,-23.358000,233.207000,-177.000000,-0.317000,167.952000,"
  [211] = "-12.733000,-23.770000,233.206000,-177.000000,-0.364000,166.178000,"
  [212] = "-14.335000,-24.242000,233.205000,-177.000000,-0.411000,164.390000,"
  [213] = "-15.934000,-24.774000,233.203000,-177.000000,-0.460000,162.586000,"
  [214] = "-17.265000,-25.265000,233.202000,-177.000000,-0.500000,161.070000,"
  [215] = "-17.284000,-25.265000,230.800000,-177.000000,-0.500000,161.072000,"
  [216] = "-17.305000,-25.264000,228.202000,-177.000000,-0.500000,161.074000,"
  [217] = "-15.971000,-24.773000,228.203000,-177.000000,-0.459000,162.590000,"
  [218] = "-14.368000,-24.241000,228.205000,-177.000000,-0.411000,164.393000,"
  [219] = "-12.762000,-23.769000,228.206000,-177.000000,-0.364000,166.181000,"
  [220] = "-11.155000,-23.357000,228.207000,-177.000000,-0.317000,167.955000,"
  [221] = "-9.545000,-23.003000,228.208000,-177.000000,-0.270000,169.717000,"
  [222] = "-7.934000,-22.705000,228.209000,-177.000000,-0.224000,171.469000,"
  [223] = "-6.322000,-22.464000,228.209000,-177.000000,-0.178000,173.213000,"
  [224] = "-4.709000,-22.278000,228.210000,-177.000000,-0.132000,174.951000,"
  [225] = "-3.095000,-22.146000,228.210000,-177.000000,-0.087000,176.685000,"
  [226] = "-1.480000,-22.070000,228.211000,-177.000000,-0.042000,178.415000,"
  [227] = "-0.135000,-22.047000,228.211000,-177.000000,-0.004000,179.856000,"
  [228] = "1.480000,-22.070000,228.211000,-177.000000,0.042000,-178.415000,"
  [229] = "3.095000,-22.146000,228.210000,-177.000000,0.087000,-176.685000,"
  [230] = "4.709000,-22.278000,228.210000,-177.000000,0.132000,-174.951000,"
  [231] = "6.322000,-22.464000,228.209000,-177.000000,0.178000,-173.213000,"
  [232] = "7.934000,-22.705000,228.209000,-177.000000,0.224000,-171.469000,"
  [233] = "9.545000,-23.003000,228.208000,-177.000000,0.270000,-169.717000,"
  [234] = "11.155000,-23.357000,228.207000,-177.000000,0.317000,-167.955000,"
  [235] = "12.763000,-23.769000,228.206000,-177.000000,0.364000,-166.181000,"
  [236] = "14.368000,-24.241000,228.205000,-177.000000,0.411000,-164.393000,"
  [237] = "15.971000,-24.773000,228.203000,-177.000000,0.459000,-162.590000,"
  [238] = "17.305000,-25.264000,228.202000,-177.000000,0.500000,-161.074000,"
  [239] = "17.328000,-25.264000,225.800000,-177.000000,0.500000,-161.072000,"
  [240] = "17.352000,-25.265000,223.202000,-177.000000,0.500000,-161.070000,"
  [241] = "15.759000,-24.685000,223.204000,-177.000000,0.452000,-162.874000,"
  [242] = "14.163000,-24.166000,223.205000,-177.000000,0.404000,-164.662000,"
  [243] = "12.565000,-23.707000,223.206000,-177.000000,0.357000,-166.434000,"
  [244] = "10.965000,-23.306000,223.207000,-177.000000,0.310000,-168.192000,"
  [245] = "9.364000,-22.962000,223.208000,-177.000000,0.264000,-169.940000,"
  [246] = "7.761000,-22.673000,223.209000,-177.000000,0.218000,-171.678000,"
  [247] = "6.156000,-22.440000,223.210000,-177.000000,0.173000,-173.409000,"
  [248] = "4.551000,-22.261000,223.210000,-177.000000,0.128000,-175.133000,"
  [249] = "2.945000,-22.137000,223.210000,-177.000000,0.082000,-176.853000,"
  [250] = "1.339000,-22.065000,223.211000,-177.000000,0.037000,-178.570000,"
  [251] = "0.268000,-22.048000,223.211000,-177.000000,0.007000,-179.714000,"
  [252] = "-1.339000,-22.065000,223.211000,-177.000000,-0.037000,178.570000,"
  [253] = "-2.945000,-22.137000,223.210000,-177.000000,-0.082000,176.853000,"
  [254] = "-4.551000,-22.261000,223.210000,-177.000000,-0.128000,175.133000,"
  [255] = "-6.156000,-22.440000,223.210000,-177.000000,-0.173000,173.409000,"
  [256] = "-7.761000,-22.673000,223.209000,-177.000000,-0.218000,171.678000,"
  [257] = "-9.364000,-22.962000,223.208000,-177.000000,-0.264000,169.940000,"
  [258] = "-10.965000,-23.306000,223.207000,-177.000000,-0.310000,168.192000,"
  [259] = "-12.565000,-23.707000,223.206000,-177.000000,-0.357000,166.434000,"
  [260] = "-14.163000,-24.166000,223.205000,-177.000000,-0.404000,164.662000,"
  [261] = "-15.759000,-24.685000,223.204000,-177.000000,-0.452000,162.874000,"
  [262] = "-17.352000,-25.265000,223.202000,-177.000000,-0.500000,161.070000,"
  [263] = "-17.371000,-25.265000,220.800000,-177.000000,-0.500000,161.072000,"
  [264] = "-17.392000,-25.264000,218.202000,-177.000000,-0.500000,161.074000,"
  [265] = "-15.795000,-24.684000,218.204000,-177.000000,-0.452000,162.878000,"
  [266] = "-14.196000,-24.166000,218.205000,-177.000000,-0.404000,164.665000,"
  [267] = "-12.594000,-23.706000,218.206000,-177.000000,-0.357000,166.436000,"
  [268] = "-10.990000,-23.305000,218.207000,-177.000000,-0.310000,168.195000,"
  [269] = "-9.385000,-22.961000,218.208000,-177.000000,-0.264000,169.942000,"
  [270] = "-7.778000,-22.673000,218.209000,-177.000000,-0.218000,171.680000,"
  [271] = "-6.170000,-22.440000,218.210000,-177.000000,-0.173000,173.410000,"
  [272] = "-4.561000,-22.261000,218.210000,-177.000000,-0.128000,175.134000,"
  [273] = "-2.952000,-22.137000,218.210000,-177.000000,-0.082000,176.854000,"
  [274] = "-1.342000,-22.065000,218.211000,-177.000000,-0.037000,178.570000,"
  [275] = "0.000000,-22.047000,218.211000,-177.000000,0.000000,180.000000,"
  [276] = "1.342000,-22.065000,218.211000,-177.000000,0.037000,-178.570000,"
  [277] = "2.952000,-22.137000,218.210000,-177.000000,0.082000,-176.854000,"
  [278] = "4.561000,-22.261000,218.210000,-177.000000,0.128000,-175.134000,"
  [279] = "6.170000,-22.440000,218.210000,-177.000000,0.173000,-173.410000,"
  [280] = "7.778000,-22.673000,218.209000,-177.000000,0.218000,-171.680000,"
  [281] = "9.385000,-22.961000,218.208000,-177.000000,0.264000,-169.942000,"
  [282] = "10.990000,-23.305000,218.207000,-177.000000,0.310000,-168.195000,"
  [283] = "12.594000,-23.706000,218.206000,-177.000000,0.357000,-166.436000,"
  [284] = "14.196000,-24.166000,218.205000,-177.000000,0.404000,-164.665000,"
  [285] = "15.795000,-24.684000,218.204000,-177.000000,0.452000,-162.878000,"
  [286] = "17.392000,-25.264000,218.202000,-177.000000,0.500000,-161.074000,"
  [287] = "17.415000,-25.264000,215.800000,-177.000000,0.500000,-161.072000,"
  [288] = "17.439000,-25.265000,213.203000,-177.000000,0.500000,-161.070000,"
  [289] = "15.838000,-24.685000,213.204000,-177.000000,0.452000,-162.874000,"
  [290] = "14.234000,-24.166000,213.205000,-177.000000,0.404000,-164.662000,"
  [291] = "12.628000,-23.707000,213.206000,-177.000000,0.357000,-166.434000,"
  [292] = "11.020000,-23.306000,213.207000,-177.000000,0.310000,-168.192000,"
  [293] = "9.410000,-22.962000,213.208000,-177.000000,0.264000,-169.940000,"
  [294] = "7.799000,-22.673000,213.209000,-177.000000,0.218000,-171.678000,"
  [295] = "6.186000,-22.440000,213.210000,-177.000000,0.173000,-173.409000,"
  [296] = "4.573000,-22.261000,213.210000,-177.000000,0.128000,-175.133000,"
  [297] = "2.959000,-22.137000,213.210000,-177.000000,0.082000,-176.853000,"
  [298] = "1.345000,-22.065000,213.211000,-177.000000,0.037000,-178.570000,"
  [299] = "0.269000,-22.048000,213.211000,-177.000000,0.007000,-179.714000,"
  [300] = "-1.345000,-22.065000,213.211000,-177.000000,-0.037000,178.570000,"
  [301] = "-2.959000,-22.137000,213.210000,-177.000000,-0.082000,176.853000,"
  [302] = "-4.573000,-22.261000,213.210000,-177.000000,-0.128000,175.133000,"
  [303] = "-6.186000,-22.440000,213.210000,-177.000000,-0.173000,173.409000,"
  [304] = "-7.799000,-22.673000,213.209000,-177.000000,-0.218000,171.678000,"
  [305] = "-9.410000,-22.962000,213.208000,-177.000000,-0.264000,169.940000,"
  [306] = "-11.020000,-23.306000,213.207000,-177.000000,-0.310000,168.192000,"
